SPLINE
SPL {X  -131.819, Y  +765.085, Z    +0.000, E1   -48.689, E3 +108359.963}
SPL {X  -153.047, Y  +721.053, Z    +0.000, E1   -34.410, E3 +108379.829}
SPL {X  -159.196, Y  +690.423, Z    +0.000, E1   -15.522, E3 +108384.926}
SPL {X  -160.000, Y  +672.957, Z    +0.000, E1    -0.766, E3 +108385.828}
SPL {X  -160.000, Y  +670.573, Z    +0.000, E1    +3.229, E3 +108385.856}
SPL {X  -160.000, Y  +665.683, Z    +0.000, E1   +13.339, E3 +108386.025}
SPL {X  -160.000, Y  +658.186, Z    +0.000, E1   +29.314, E3 +108386.629}
SPL {X  -160.000, Y  +642.169, Z    +0.000, E1   +52.097, E3 +108389.155}
SPL {X  -160.000, Y  +581.106, Z    +0.000, E1   +69.111, E3 +108410.027}
SPL {X  -160.000, Y  +418.281, Z    +0.000, E1   +71.209, E3 +108501.377}
SPL {X  -153.877, Y  +341.861, Z    +0.000, E1   +74.632, E3 +108514.790}
SPL {X  -152.649, Y  +337.758, Z    +0.000, E1   +72.728, E3 +108536.453}
SPL {X  -150.568, Y  +331.578, Z    +0.000, E1   +70.963, E3 +108556.379}
SPL {X  -147.367, Y  +323.387, Z    +0.000, E1   +69.846, E3 +108570.999}
SPL {X  -143.458, Y  +314.849, Z    +0.000, E1   +69.330, E3 +108580.881}
SPL {X  -137.919, Y  +304.592, Z    +0.000, E1   +68.645, E3 +108593.170}
SPL {X  -132.252, Y  +295.648, Z    +0.000, E1   +67.759, E3 +108604.485}
SPL {X  -127.852, Y  +289.504, Z    +0.000, E1   +67.080, E3 +108612.317}
SPL {X  -124.264, Y  +284.911, Z    +0.000, E1   +66.468, E3 +108618.213}
SPL {X   -87.531, Y  +251.766, Z    +0.000, E1   +54.242, E3 +108746.530}
ENDSPLINE

SPLINE
SPL {X  -130.414, Y  +293.006, Z    +0.000, E1   +48.816, E3 +108895.142}
SPL {X  -151.093, Y  +333.061, Z    +0.000, E1   +36.955, E3 +108916.423}
SPL {X  -158.896, Y  +366.939, Z    +0.000, E1   +17.535, E3 +108922.962}
SPL {X  -160.000, Y  +387.267, Z    +0.000, E1    +0.577, E3 +108924.152}
SPL {X  -160.000, Y  +391.471, Z    +0.000, E1    -7.208, E3 +108924.233}
SPL {X  -160.000, Y  +398.523, Z    +0.000, E1   -22.265, E3 +108924.645}
SPL {X  -160.000, Y  +411.325, Z    +0.000, E1   -44.857, E3 +108926.311}
SPL {X  -160.000, Y  +459.786, Z    +0.000, E1   -66.828, E3 +108941.704}
SPL {X  -160.000, Y  +650.407, Z    +0.000, E1   -71.387, E3 +109044.361}
SPL {X  -159.770, Y  +682.971, Z    +0.000, E1   -71.362, E3 +109067.936}
SPL {X  -156.288, Y  +708.665, Z    +0.000, E1   -70.996, E3 +109089.946}
SPL {X  -150.837, Y  +727.770, Z    +0.000, E1   -70.337, E3 +109109.280}
SPL {X  -144.661, Y  +742.760, Z    +0.000, E1   -69.570, E3 +109126.038}
SPL {X  -137.606, Y  +756.037, Z    +0.000, E1   -68.631, E3 +109142.003}
SPL {X  -131.907, Y  +764.957, Z    +0.000, E1   -67.736, E3 +109153.298}
SPL {X  -127.608, Y  +770.921, Z    +0.000, E1   -67.067, E3 +109160.917}
SPL {X  -124.072, Y  +775.426, Z    +0.000, E1   -66.459, E3 +109166.697}
SPL {X   -86.375, Y  +809.082, Z    +0.000, E1   -54.606, E3 +109291.027}
ENDSPLINE

SPLINE
SPL {X  -131.819, Y  +765.085, Z    +0.000, E1   -48.689, E3 +109446.921}
SPL {X  -153.047, Y  +721.053, Z    +0.000, E1   -34.410, E3 +109466.787}
SPL {X  -159.196, Y  +690.423, Z    +0.000, E1   -15.522, E3 +109471.883}
SPL {X  -160.000, Y  +672.957, Z    +0.000, E1    -0.766, E3 +109472.785}
SPL {X  -160.000, Y  +670.573, Z    +0.000, E1    +3.229, E3 +109472.813}
SPL {X  -160.000, Y  +665.683, Z    +0.000, E1   +13.339, E3 +109472.982}
SPL {X  -160.000, Y  +658.186, Z    +0.000, E1   +29.314, E3 +109473.586}
SPL {X  -160.000, Y  +642.169, Z    +0.000, E1   +52.097, E3 +109476.112}
SPL {X  -160.000, Y  +581.106, Z    +0.000, E1   +69.111, E3 +109496.984}
SPL {X  -160.000, Y  +418.281, Z    +0.000, E1   +71.209, E3 +109588.334}
SPL {X  -153.877, Y  +341.861, Z    +0.000, E1   +74.632, E3 +109601.747}
SPL {X  -152.649, Y  +337.758, Z    +0.000, E1   +72.728, E3 +109623.410}
SPL {X  -150.568, Y  +331.578, Z    +0.000, E1   +70.963, E3 +109643.336}
SPL {X  -147.367, Y  +323.387, Z    +0.000, E1   +69.846, E3 +109657.956}
SPL {X  -143.458, Y  +314.849, Z    +0.000, E1   +69.330, E3 +109667.839}
SPL {X  -137.919, Y  +304.592, Z    +0.000, E1   +68.645, E3 +109680.127}
SPL {X  -132.252, Y  +295.648, Z    +0.000, E1   +67.759, E3 +109691.442}
SPL {X  -127.852, Y  +289.504, Z    +0.000, E1   +67.080, E3 +109699.274}
SPL {X  -124.264, Y  +284.911, Z    +0.000, E1   +66.468, E3 +109705.170}
SPL {X   -87.531, Y  +251.766, Z    +0.000, E1   +54.242, E3 +109833.487}
ENDSPLINE

SPLINE
SPL {X  -130.414, Y  +293.006, Z    +0.000, E1   +48.816, E3 +109982.099}
SPL {X  -151.093, Y  +333.061, Z    +0.000, E1   +36.955, E3 +110003.380}
SPL {X  -158.896, Y  +366.939, Z    +0.000, E1   +17.535, E3 +110009.919}
SPL {X  -160.000, Y  +387.267, Z    +0.000, E1    +0.577, E3 +110011.109}
SPL {X  -160.000, Y  +391.471, Z    +0.000, E1    -7.208, E3 +110011.190}
SPL {X  -160.000, Y  +398.523, Z    +0.000, E1   -22.265, E3 +110011.602}
SPL {X  -160.000, Y  +411.325, Z    +0.000, E1   -44.857, E3 +110013.268}
SPL {X  -160.000, Y  +459.786, Z    +0.000, E1   -66.828, E3 +110028.661}
SPL {X  -160.000, Y  +650.407, Z    +0.000, E1   -71.387, E3 +110131.318}
SPL {X  -159.770, Y  +682.971, Z    +0.000, E1   -71.362, E3 +110154.893}
SPL {X  -156.288, Y  +708.665, Z    +0.000, E1   -70.996, E3 +110176.903}
SPL {X  -150.837, Y  +727.770, Z    +0.000, E1   -70.337, E3 +110196.237}
SPL {X  -144.661, Y  +742.760, Z    +0.000, E1   -69.570, E3 +110212.995}
SPL {X  -137.606, Y  +756.037, Z    +0.000, E1   -68.631, E3 +110228.960}
SPL {X  -131.907, Y  +764.957, Z    +0.000, E1   -67.736, E3 +110240.255}
SPL {X  -127.608, Y  +770.921, Z    +0.000, E1   -67.067, E3 +110247.874}
SPL {X  -124.072, Y  +775.426, Z    +0.000, E1   -66.459, E3 +110253.654}
SPL {X   -86.375, Y  +809.082, Z    +0.000, E1   -54.606, E3 +110377.984}
ENDSPLINE

SPLINE
SPL {X  -131.819, Y  +765.085, Z    +0.000, E1   -48.689, E3 +110533.878}
SPL {X  -153.047, Y  +721.053, Z    +0.000, E1   -34.410, E3 +110553.744}
SPL {X  -159.196, Y  +690.423, Z    +0.000, E1   -15.522, E3 +110558.840}
SPL {X  -160.000, Y  +672.957, Z    +0.000, E1    -0.766, E3 +110559.742}
SPL {X  -160.000, Y  +670.573, Z    +0.000, E1    +3.229, E3 +110559.770}
SPL {X  -160.000, Y  +665.683, Z    +0.000, E1   +13.339, E3 +110559.939}
SPL {X  -160.000, Y  +658.186, Z    +0.000, E1   +29.314, E3 +110560.544}
SPL {X  -160.000, Y  +642.169, Z    +0.000, E1   +52.097, E3 +110563.069}
SPL {X  -160.000, Y  +581.106, Z    +0.000, E1   +69.111, E3 +110583.941}
SPL {X  -160.000, Y  +418.281, Z    +0.000, E1   +71.209, E3 +110675.291}
SPL {X  -153.877, Y  +341.861, Z    +0.000, E1   +74.632, E3 +110688.704}
SPL {X  -152.649, Y  +337.758, Z    +0.000, E1   +72.728, E3 +110710.367}
SPL {X  -150.568, Y  +331.578, Z    +0.000, E1   +70.963, E3 +110730.293}
SPL {X  -147.367, Y  +323.387, Z    +0.000, E1   +69.846, E3 +110744.913}
SPL {X  -143.458, Y  +314.849, Z    +0.000, E1   +69.330, E3 +110754.796}
SPL {X  -137.919, Y  +304.592, Z    +0.000, E1   +68.645, E3 +110767.084}
SPL {X  -132.252, Y  +295.648, Z    +0.000, E1   +67.759, E3 +110778.399}
SPL {X  -127.852, Y  +289.504, Z    +0.000, E1   +67.080, E3 +110786.231}
SPL {X  -124.264, Y  +284.911, Z    +0.000, E1   +66.468, E3 +110792.127}
SPL {X   -87.531, Y  +251.766, Z    +0.000, E1   +54.242, E3 +110920.444}
ENDSPLINE

SPLINE
SPL {X  -130.414, Y  +293.006, Z    +0.000, E1   +48.816, E3 +111069.056}
SPL {X  -151.093, Y  +333.061, Z    +0.000, E1   +36.955, E3 +111090.337}
SPL {X  -158.896, Y  +366.939, Z    +0.000, E1   +17.535, E3 +111096.877}
SPL {X  -160.000, Y  +387.267, Z    +0.000, E1    +0.577, E3 +111098.066}
SPL {X  -160.000, Y  +391.471, Z    +0.000, E1    -7.208, E3 +111098.147}
SPL {X  -160.000, Y  +398.523, Z    +0.000, E1   -22.265, E3 +111098.559}
SPL {X  -160.000, Y  +411.325, Z    +0.000, E1   -44.857, E3 +111100.225}
SPL {X  -160.000, Y  +459.786, Z    +0.000, E1   -66.828, E3 +111115.618}
SPL {X  -160.000, Y  +650.407, Z    +0.000, E1   -71.387, E3 +111218.275}
SPL {X  -159.770, Y  +682.971, Z    +0.000, E1   -71.362, E3 +111241.850}
SPL {X  -156.288, Y  +708.665, Z    +0.000, E1   -70.996, E3 +111263.861}
SPL {X  -150.837, Y  +727.770, Z    +0.000, E1   -70.337, E3 +111283.194}
SPL {X  -144.661, Y  +742.760, Z    +0.000, E1   -69.570, E3 +111299.953}
SPL {X  -137.606, Y  +756.037, Z    +0.000, E1   -68.631, E3 +111315.917}
SPL {X  -131.907, Y  +764.957, Z    +0.000, E1   -67.736, E3 +111327.212}
SPL {X  -127.608, Y  +770.921, Z    +0.000, E1   -67.067, E3 +111334.831}
SPL {X  -124.072, Y  +775.426, Z    +0.000, E1   -66.459, E3 +111340.611}
SPL {X   -86.375, Y  +809.082, Z    +0.000, E1   -54.606, E3 +111464.941}
ENDSPLINE

SPLINE
SPL {X  -131.819, Y  +765.085, Z    +0.000, E1   -48.689, E3 +111620.835}
SPL {X  -153.047, Y  +721.053, Z    +0.000, E1   -34.410, E3 +111640.701}
SPL {X  -159.196, Y  +690.423, Z    +0.000, E1   -15.522, E3 +111645.797}
SPL {X  -160.000, Y  +672.957, Z    +0.000, E1    -0.766, E3 +111646.699}
SPL {X  -160.000, Y  +670.573, Z    +0.000, E1    +3.229, E3 +111646.727}
SPL {X  -160.000, Y  +665.683, Z    +0.000, E1   +13.339, E3 +111646.896}
SPL {X  -160.000, Y  +658.186, Z    +0.000, E1   +29.314, E3 +111647.501}
SPL {X  -160.000, Y  +642.169, Z    +0.000, E1   +52.097, E3 +111650.026}
SPL {X  -160.000, Y  +581.106, Z    +0.000, E1   +69.111, E3 +111670.898}
SPL {X  -160.000, Y  +418.281, Z    +0.000, E1   +71.209, E3 +111762.248}
SPL {X  -153.877, Y  +341.861, Z    +0.000, E1   +74.632, E3 +111775.662}
SPL {X  -152.649, Y  +337.758, Z    +0.000, E1   +72.728, E3 +111797.324}
SPL {X  -150.568, Y  +331.578, Z    +0.000, E1   +70.963, E3 +111817.250}
SPL {X  -147.367, Y  +323.387, Z    +0.000, E1   +69.846, E3 +111831.870}
SPL {X  -143.458, Y  +314.849, Z    +0.000, E1   +69.330, E3 +111841.753}
SPL {X  -137.919, Y  +304.592, Z    +0.000, E1   +68.645, E3 +111854.041}
SPL {X  -132.252, Y  +295.648, Z    +0.000, E1   +67.759, E3 +111865.356}
SPL {X  -127.852, Y  +289.504, Z    +0.000, E1   +67.080, E3 +111873.188}
SPL {X  -124.264, Y  +284.911, Z    +0.000, E1   +66.468, E3 +111879.084}
SPL {X   -87.531, Y  +251.766, Z    +0.000, E1   +54.242, E3 +112007.401}
ENDSPLINE

SPLINE
SPL {X  -130.414, Y  +293.006, Z    +0.000, E1   +48.816, E3 +112156.013}
SPL {X  -151.093, Y  +333.061, Z    +0.000, E1   +36.955, E3 +112177.294}
SPL {X  -158.896, Y  +366.939, Z    +0.000, E1   +17.535, E3 +112183.834}
SPL {X  -160.000, Y  +387.267, Z    +0.000, E1    +0.577, E3 +112185.024}
SPL {X  -160.000, Y  +391.471, Z    +0.000, E1    -7.208, E3 +112185.104}
SPL {X  -160.000, Y  +398.523, Z    +0.000, E1   -22.265, E3 +112185.516}
SPL {X  -160.000, Y  +411.325, Z    +0.000, E1   -44.857, E3 +112187.182}
SPL {X  -160.000, Y  +459.786, Z    +0.000, E1   -66.828, E3 +112202.575}
SPL {X  -160.000, Y  +650.407, Z    +0.000, E1   -71.387, E3 +112305.232}
SPL {X  -159.770, Y  +682.971, Z    +0.000, E1   -71.362, E3 +112328.807}
SPL {X  -156.288, Y  +708.665, Z    +0.000, E1   -70.996, E3 +112350.818}
SPL {X  -150.837, Y  +727.770, Z    +0.000, E1   -70.337, E3 +112370.151}
SPL {X  -144.661, Y  +742.760, Z    +0.000, E1   -69.570, E3 +112386.910}
SPL {X  -137.606, Y  +756.037, Z    +0.000, E1   -68.631, E3 +112402.874}
SPL {X  -131.907, Y  +764.957, Z    +0.000, E1   -67.736, E3 +112414.169}
SPL {X  -127.608, Y  +770.921, Z    +0.000, E1   -67.067, E3 +112421.788}
SPL {X  -124.072, Y  +775.426, Z    +0.000, E1   -66.459, E3 +112427.568}
SPL {X   -86.375, Y  +809.082, Z    +0.000, E1   -54.606, E3 +112551.898}
ENDSPLINE

SPLINE
SPL {X  -131.819, Y  +765.085, Z    +0.000, E1   -48.689, E3 +112707.792}
SPL {X  -153.047, Y  +721.053, Z    +0.000, E1   -34.410, E3 +112727.658}
SPL {X  -159.196, Y  +690.423, Z    +0.000, E1   -15.522, E3 +112732.754}
SPL {X  -160.000, Y  +672.957, Z    +0.000, E1    -0.766, E3 +112733.656}
SPL {X  -160.000, Y  +670.573, Z    +0.000, E1    +3.229, E3 +112733.684}
SPL {X  -160.000, Y  +665.683, Z    +0.000, E1   +13.339, E3 +112733.854}
SPL {X  -160.000, Y  +658.186, Z    +0.000, E1   +29.314, E3 +112734.458}
SPL {X  -160.000, Y  +642.169, Z    +0.000, E1   +52.097, E3 +112736.983}
SPL {X  -160.000, Y  +581.106, Z    +0.000, E1   +69.111, E3 +112757.856}
SPL {X  -160.000, Y  +418.281, Z    +0.000, E1   +71.209, E3 +112849.205}
SPL {X  -153.877, Y  +341.861, Z    +0.000, E1   +74.632, E3 +112862.619}
SPL {X  -152.649, Y  +337.758, Z    +0.000, E1   +72.728, E3 +112884.281}
SPL {X  -150.568, Y  +331.578, Z    +0.000, E1   +70.963, E3 +112904.207}
SPL {X  -147.367, Y  +323.387, Z    +0.000, E1   +69.846, E3 +112918.828}
SPL {X  -143.458, Y  +314.849, Z    +0.000, E1   +69.330, E3 +112928.710}
SPL {X  -137.919, Y  +304.592, Z    +0.000, E1   +68.645, E3 +112940.999}
SPL {X  -132.252, Y  +295.648, Z    +0.000, E1   +67.759, E3 +112952.313}
SPL {X  -127.852, Y  +289.504, Z    +0.000, E1   +67.080, E3 +112960.146}
SPL {X  -124.264, Y  +284.911, Z    +0.000, E1   +66.468, E3 +112966.041}
SPL {X   -87.531, Y  +251.766, Z    +0.000, E1   +54.242, E3 +113094.358}
ENDSPLINE

SPLINE
SPL {X  -130.414, Y  +293.006, Z    +0.000, E1   +48.816, E3 +113242.971}
SPL {X  -151.093, Y  +333.061, Z    +0.000, E1   +36.955, E3 +113264.251}
SPL {X  -158.896, Y  +366.939, Z    +0.000, E1   +17.535, E3 +113270.791}
SPL {X  -160.000, Y  +387.267, Z    +0.000, E1    +0.577, E3 +113271.981}
SPL {X  -160.000, Y  +391.471, Z    +0.000, E1    -7.208, E3 +113272.062}
SPL {X  -160.000, Y  +398.523, Z    +0.000, E1   -22.265, E3 +113272.473}
SPL {X  -160.000, Y  +411.325, Z    +0.000, E1   -44.857, E3 +113274.139}
SPL {X  -160.000, Y  +459.786, Z    +0.000, E1   -66.828, E3 +113289.532}
SPL {X  -160.000, Y  +650.407, Z    +0.000, E1   -71.387, E3 +113392.189}
SPL {X  -159.770, Y  +682.971, Z    +0.000, E1   -71.362, E3 +113415.765}
SPL {X  -156.288, Y  +708.665, Z    +0.000, E1   -70.996, E3 +113437.775}
SPL {X  -150.837, Y  +727.770, Z    +0.000, E1   -70.337, E3 +113457.108}
SPL {X  -144.661, Y  +742.760, Z    +0.000, E1   -69.570, E3 +113473.867}
SPL {X  -137.606, Y  +756.037, Z    +0.000, E1   -68.631, E3 +113489.831}
SPL {X  -131.907, Y  +764.957, Z    +0.000, E1   -67.736, E3 +113501.126}
SPL {X  -127.608, Y  +770.921, Z    +0.000, E1   -67.067, E3 +113508.745}
SPL {X  -124.072, Y  +775.426, Z    +0.000, E1   -66.459, E3 +113514.525}
SPL {X   -86.375, Y  +809.082, Z    +0.000, E1   -54.606, E3 +113638.856}
ENDSPLINE

SPLINE
SPL {X  -131.819, Y  +765.085, Z    +0.000, E1   -48.689, E3 +113794.749}
SPL {X  -153.047, Y  +721.053, Z    +0.000, E1   -34.410, E3 +113814.615}
SPL {X  -159.196, Y  +690.423, Z    +0.000, E1   -15.522, E3 +113819.711}
SPL {X  -160.000, Y  +672.957, Z    +0.000, E1    -0.766, E3 +113820.613}
SPL {X  -160.000, Y  +670.573, Z    +0.000, E1    +3.229, E3 +113820.641}
SPL {X  -160.000, Y  +665.683, Z    +0.000, E1   +13.339, E3 +113820.811}
SPL {X  -160.000, Y  +658.186, Z    +0.000, E1   +29.314, E3 +113821.415}
SPL {X  -160.000, Y  +642.169, Z    +0.000, E1   +52.097, E3 +113823.940}
SPL {X  -160.000, Y  +581.106, Z    +0.000, E1   +69.111, E3 +113844.813}
SPL {X  -160.000, Y  +418.281, Z    +0.000, E1   +71.209, E3 +113936.162}
SPL {X  -153.877, Y  +341.861, Z    +0.000, E1   +74.632, E3 +113949.576}
SPL {X  -152.649, Y  +337.758, Z    +0.000, E1   +72.728, E3 +113971.238}
SPL {X  -150.568, Y  +331.578, Z    +0.000, E1   +70.963, E3 +113991.164}
SPL {X  -147.367, Y  +323.387, Z    +0.000, E1   +69.846, E3 +114005.785}
SPL {X  -143.458, Y  +314.849, Z    +0.000, E1   +69.330, E3 +114015.667}
SPL {X  -137.919, Y  +304.592, Z    +0.000, E1   +68.645, E3 +114027.956}
SPL {X  -132.252, Y  +295.648, Z    +0.000, E1   +67.759, E3 +114039.270}
SPL {X  -127.852, Y  +289.504, Z    +0.000, E1   +67.080, E3 +114047.103}
SPL {X  -124.264, Y  +284.911, Z    +0.000, E1   +66.468, E3 +114052.999}
SPL {X   -87.531, Y  +251.766, Z    +0.000, E1   +54.242, E3 +114181.315}
ENDSPLINE

SPLINE
SPL {X  -130.414, Y  +293.006, Z    +0.000, E1   +48.816, E3 +114329.928}
SPL {X  -151.093, Y  +333.061, Z    +0.000, E1   +36.955, E3 +114351.208}
SPL {X  -158.896, Y  +366.939, Z    +0.000, E1   +17.535, E3 +114357.748}
SPL {X  -160.000, Y  +387.267, Z    +0.000, E1    +0.577, E3 +114358.938}
SPL {X  -160.000, Y  +391.471, Z    +0.000, E1    -7.208, E3 +114359.019}
SPL {X  -160.000, Y  +398.523, Z    +0.000, E1   -22.265, E3 +114359.431}
SPL {X  -160.000, Y  +411.325, Z    +0.000, E1   -44.857, E3 +114361.096}
SPL {X  -160.000, Y  +459.786, Z    +0.000, E1   -66.828, E3 +114376.489}
SPL {X  -160.000, Y  +650.407, Z    +0.000, E1   -71.387, E3 +114479.146}
SPL {X  -159.770, Y  +682.971, Z    +0.000, E1   -71.362, E3 +114502.722}
SPL {X  -156.288, Y  +708.665, Z    +0.000, E1   -70.996, E3 +114524.732}
SPL {X  -150.837, Y  +727.770, Z    +0.000, E1   -70.337, E3 +114544.066}
SPL {X  -144.661, Y  +742.760, Z    +0.000, E1   -69.570, E3 +114560.824}
SPL {X  -137.606, Y  +756.037, Z    +0.000, E1   -68.631, E3 +114576.789}
SPL {X  -131.907, Y  +764.957, Z    +0.000, E1   -67.736, E3 +114588.084}
SPL {X  -127.608, Y  +770.921, Z    +0.000, E1   -67.067, E3 +114595.702}
SPL {X  -124.072, Y  +775.426, Z    +0.000, E1   -66.459, E3 +114601.482}
SPL {X   -86.375, Y  +809.082, Z    +0.000, E1   -54.606, E3 +114725.813}
ENDSPLINE

SPLINE
SPL {X  -131.819, Y  +765.085, Z    +0.000, E1   -48.689, E3 +114881.706}
SPL {X  -153.047, Y  +721.053, Z    +0.000, E1   -34.410, E3 +114901.572}
SPL {X  -159.196, Y  +690.423, Z    +0.000, E1   -15.522, E3 +114906.669}
SPL {X  -160.000, Y  +672.957, Z    +0.000, E1    -0.766, E3 +114907.570}
SPL {X  -160.000, Y  +670.573, Z    +0.000, E1    +3.229, E3 +114907.599}
SPL {X  -160.000, Y  +665.683, Z    +0.000, E1   +13.339, E3 +114907.768}
SPL {X  -160.000, Y  +658.186, Z    +0.000, E1   +29.314, E3 +114908.372}
SPL {X  -160.000, Y  +642.169, Z    +0.000, E1   +52.097, E3 +114910.898}
SPL {X  -160.000, Y  +581.106, Z    +0.000, E1   +69.111, E3 +114931.770}
SPL {X  -160.000, Y  +418.281, Z    +0.000, E1   +71.209, E3 +115023.119}
SPL {X  -153.877, Y  +341.861, Z    +0.000, E1   +74.632, E3 +115036.533}
SPL {X  -152.649, Y  +337.758, Z    +0.000, E1   +72.728, E3 +115058.196}
SPL {X  -150.568, Y  +331.578, Z    +0.000, E1   +70.963, E3 +115078.121}
SPL {X  -147.367, Y  +323.387, Z    +0.000, E1   +69.846, E3 +115092.742}
SPL {X  -143.458, Y  +314.849, Z    +0.000, E1   +69.330, E3 +115102.624}
SPL {X  -137.919, Y  +304.592, Z    +0.000, E1   +68.645, E3 +115114.913}
SPL {X  -132.252, Y  +295.648, Z    +0.000, E1   +67.759, E3 +115126.228}
SPL {X  -127.852, Y  +289.504, Z    +0.000, E1   +67.080, E3 +115134.060}
SPL {X  -124.264, Y  +284.911, Z    +0.000, E1   +66.468, E3 +115139.956}
SPL {X   -87.531, Y  +251.766, Z    +0.000, E1   +54.242, E3 +115268.272}
ENDSPLINE

SPLINE
SPL {X  -130.414, Y  +293.006, Z    +0.000, E1   +48.816, E3 +115416.885}
SPL {X  -151.093, Y  +333.061, Z    +0.000, E1   +36.955, E3 +115438.165}
SPL {X  -158.896, Y  +366.939, Z    +0.000, E1   +17.535, E3 +115444.705}
SPL {X  -160.000, Y  +387.267, Z    +0.000, E1    +0.577, E3 +115445.895}
SPL {X  -160.000, Y  +391.471, Z    +0.000, E1    -7.208, E3 +115445.976}
SPL {X  -160.000, Y  +398.523, Z    +0.000, E1   -22.265, E3 +115446.388}
SPL {X  -160.000, Y  +411.325, Z    +0.000, E1   -44.857, E3 +115448.054}
SPL {X  -160.000, Y  +459.786, Z    +0.000, E1   -66.828, E3 +115463.446}
SPL {X  -160.000, Y  +650.407, Z    +0.000, E1   -71.387, E3 +115566.103}
SPL {X  -159.770, Y  +682.971, Z    +0.000, E1   -71.362, E3 +115589.679}
SPL {X  -156.288, Y  +708.665, Z    +0.000, E1   -70.996, E3 +115611.689}
SPL {X  -150.837, Y  +727.770, Z    +0.000, E1   -70.337, E3 +115631.023}
SPL {X  -144.661, Y  +742.760, Z    +0.000, E1   -69.570, E3 +115647.781}
SPL {X  -137.606, Y  +756.037, Z    +0.000, E1   -68.631, E3 +115663.746}
SPL {X  -131.907, Y  +764.957, Z    +0.000, E1   -67.736, E3 +115675.041}
SPL {X  -127.608, Y  +770.921, Z    +0.000, E1   -67.067, E3 +115682.659}
SPL {X  -124.072, Y  +775.426, Z    +0.000, E1   -66.459, E3 +115688.440}
SPL {X   -86.375, Y  +809.082, Z    +0.000, E1   -54.606, E3 +115812.770}
ENDSPLINE

SPLINE
SPL {X  -131.819, Y  +765.085, Z    +0.000, E1   -48.689, E3 +115968.663}
SPL {X  -153.047, Y  +721.053, Z    +0.000, E1   -34.410, E3 +115988.529}
SPL {X  -159.196, Y  +690.423, Z    +0.000, E1   -15.522, E3 +115993.626}
SPL {X  -160.000, Y  +672.957, Z    +0.000, E1    -0.766, E3 +115994.528}
SPL {X  -160.000, Y  +670.573, Z    +0.000, E1    +3.229, E3 +115994.556}
SPL {X  -160.000, Y  +665.683, Z    +0.000, E1   +13.339, E3 +115994.725}
SPL {X  -160.000, Y  +658.186, Z    +0.000, E1   +29.314, E3 +115995.329}
SPL {X  -160.000, Y  +642.169, Z    +0.000, E1   +52.097, E3 +115997.855}
SPL {X  -160.000, Y  +581.106, Z    +0.000, E1   +69.111, E3 +116018.727}
SPL {X  -160.000, Y  +418.281, Z    +0.000, E1   +71.209, E3 +116110.076}
SPL {X  -153.877, Y  +341.861, Z    +0.000, E1   +74.632, E3 +116123.490}
SPL {X  -152.649, Y  +337.758, Z    +0.000, E1   +72.728, E3 +116145.153}
SPL {X  -150.568, Y  +331.578, Z    +0.000, E1   +70.963, E3 +116165.079}
SPL {X  -147.367, Y  +323.387, Z    +0.000, E1   +69.846, E3 +116179.699}
SPL {X  -143.458, Y  +314.849, Z    +0.000, E1   +69.330, E3 +116189.581}
SPL {X  -137.919, Y  +304.592, Z    +0.000, E1   +68.645, E3 +116201.870}
SPL {X  -132.252, Y  +295.648, Z    +0.000, E1   +67.759, E3 +116213.185}
SPL {X  -127.852, Y  +289.504, Z    +0.000, E1   +67.080, E3 +116221.017}
SPL {X  -124.264, Y  +284.911, Z    +0.000, E1   +66.468, E3 +116226.913}
SPL {X   -87.531, Y  +251.766, Z    +0.000, E1   +54.242, E3 +116355.229}
ENDSPLINE

SPLINE
SPL {X  -130.414, Y  +293.006, Z    +0.000, E1   +48.816, E3 +116503.842}
SPL {X  -151.093, Y  +333.061, Z    +0.000, E1   +36.955, E3 +116525.122}
SPL {X  -158.896, Y  +366.939, Z    +0.000, E1   +17.535, E3 +116531.662}
SPL {X  -160.000, Y  +387.267, Z    +0.000, E1    +0.577, E3 +116532.852}
SPL {X  -160.000, Y  +391.471, Z    +0.000, E1    -7.208, E3 +116532.933}
SPL {X  -160.000, Y  +398.523, Z    +0.000, E1   -22.265, E3 +116533.345}
SPL {X  -160.000, Y  +411.325, Z    +0.000, E1   -44.857, E3 +116535.011}
SPL {X  -160.000, Y  +459.786, Z    +0.000, E1   -66.828, E3 +116550.403}
SPL {X  -160.000, Y  +650.407, Z    +0.000, E1   -71.387, E3 +116653.060}
SPL {X  -159.770, Y  +682.971, Z    +0.000, E1   -71.362, E3 +116676.636}
SPL {X  -156.288, Y  +708.665, Z    +0.000, E1   -70.996, E3 +116698.646}
SPL {X  -150.837, Y  +727.770, Z    +0.000, E1   -70.337, E3 +116717.980}
SPL {X  -144.661, Y  +742.760, Z    +0.000, E1   -69.570, E3 +116734.738}
SPL {X  -137.606, Y  +756.037, Z    +0.000, E1   -68.631, E3 +116750.703}
SPL {X  -131.907, Y  +764.957, Z    +0.000, E1   -67.736, E3 +116761.998}
SPL {X  -127.608, Y  +770.921, Z    +0.000, E1   -67.067, E3 +116769.616}
SPL {X  -124.072, Y  +775.426, Z    +0.000, E1   -66.459, E3 +116775.397}
SPL {X   -86.375, Y  +809.082, Z    +0.000, E1   -54.606, E3 +116899.727}
ENDSPLINE

SPLINE
SPL {X  -131.819, Y  +765.085, Z    +0.000, E1   -48.689, E3 +117055.620}
SPL {X  -153.047, Y  +721.053, Z    +0.000, E1   -34.410, E3 +117075.486}
SPL {X  -159.196, Y  +690.423, Z    +0.000, E1   -15.522, E3 +117080.583}
SPL {X  -160.000, Y  +672.957, Z    +0.000, E1    -0.766, E3 +117081.485}
SPL {X  -160.000, Y  +670.573, Z    +0.000, E1    +3.229, E3 +117081.513}
SPL {X  -160.000, Y  +665.683, Z    +0.000, E1   +13.339, E3 +117081.682}
SPL {X  -160.000, Y  +658.186, Z    +0.000, E1   +29.314, E3 +117082.286}
SPL {X  -160.000, Y  +642.169, Z    +0.000, E1   +52.097, E3 +117084.812}
SPL {X  -160.000, Y  +581.106, Z    +0.000, E1   +69.111, E3 +117105.684}
SPL {X  -160.000, Y  +418.281, Z    +0.000, E1   +71.209, E3 +117197.034}
SPL {X  -153.877, Y  +341.861, Z    +0.000, E1   +74.632, E3 +117210.447}
SPL {X  -152.649, Y  +337.758, Z    +0.000, E1   +72.728, E3 +117232.110}
SPL {X  -150.568, Y  +331.578, Z    +0.000, E1   +70.963, E3 +117252.036}
SPL {X  -147.367, Y  +323.387, Z    +0.000, E1   +69.846, E3 +117266.656}
SPL {X  -143.458, Y  +314.849, Z    +0.000, E1   +69.330, E3 +117276.538}
SPL {X  -137.919, Y  +304.592, Z    +0.000, E1   +68.645, E3 +117288.827}
SPL {X  -132.252, Y  +295.648, Z    +0.000, E1   +67.759, E3 +117300.142}
SPL {X  -127.852, Y  +289.504, Z    +0.000, E1   +67.080, E3 +117307.974}
SPL {X  -124.264, Y  +284.911, Z    +0.000, E1   +66.468, E3 +117313.870}
SPL {X   -87.531, Y  +251.766, Z    +0.000, E1   +54.242, E3 +117442.187}
ENDSPLINE

SPLINE
SPL {X  -130.414, Y  +293.006, Z    +0.000, E1   +48.816, E3 +117590.799}
SPL {X  -151.093, Y  +333.061, Z    +0.000, E1   +36.955, E3 +117612.080}
SPL {X  -158.896, Y  +366.939, Z    +0.000, E1   +17.535, E3 +117618.619}
SPL {X  -160.000, Y  +387.267, Z    +0.000, E1    +0.577, E3 +117619.809}
SPL {X  -160.000, Y  +391.471, Z    +0.000, E1    -7.208, E3 +117619.890}
SPL {X  -160.000, Y  +398.523, Z    +0.000, E1   -22.265, E3 +117620.302}
SPL {X  -160.000, Y  +411.325, Z    +0.000, E1   -44.857, E3 +117621.968}
SPL {X  -160.000, Y  +459.786, Z    +0.000, E1   -66.828, E3 +117637.361}
SPL {X  -160.000, Y  +650.407, Z    +0.000, E1   -71.387, E3 +117740.018}
SPL {X  -159.770, Y  +682.971, Z    +0.000, E1   -71.362, E3 +117763.593}
SPL {X  -156.288, Y  +708.665, Z    +0.000, E1   -70.996, E3 +117785.603}
SPL {X  -150.837, Y  +727.770, Z    +0.000, E1   -70.337, E3 +117804.937}
SPL {X  -144.661, Y  +742.760, Z    +0.000, E1   -69.570, E3 +117821.695}
SPL {X  -137.606, Y  +756.037, Z    +0.000, E1   -68.631, E3 +117837.660}
SPL {X  -131.907, Y  +764.957, Z    +0.000, E1   -67.736, E3 +117848.955}
SPL {X  -127.608, Y  +770.921, Z    +0.000, E1   -67.067, E3 +117856.573}
SPL {X  -124.072, Y  +775.426, Z    +0.000, E1   -66.459, E3 +117862.354}
SPL {X   -86.375, Y  +809.082, Z    +0.000, E1   -54.606, E3 +117986.684}
ENDSPLINE

SPLINE
SPL {X  -131.819, Y  +765.085, Z    +0.000, E1   -48.689, E3 +118142.577}
SPL {X  -153.047, Y  +721.053, Z    +0.000, E1   -34.410, E3 +118162.443}
SPL {X  -159.196, Y  +690.423, Z    +0.000, E1   -15.522, E3 +118167.540}
SPL {X  -160.000, Y  +672.957, Z    +0.000, E1    -0.766, E3 +118168.442}
SPL {X  -160.000, Y  +670.573, Z    +0.000, E1    +3.229, E3 +118168.470}
SPL {X  -160.000, Y  +665.683, Z    +0.000, E1   +13.339, E3 +118168.639}
SPL {X  -160.000, Y  +658.186, Z    +0.000, E1   +29.314, E3 +118169.243}
SPL {X  -160.000, Y  +642.169, Z    +0.000, E1   +52.097, E3 +118171.769}
SPL {X  -160.000, Y  +581.106, Z    +0.000, E1   +69.111, E3 +118192.641}
SPL {X  -160.000, Y  +418.281, Z    +0.000, E1   +71.209, E3 +118283.991}
SPL {X  -153.877, Y  +341.861, Z    +0.000, E1   +74.632, E3 +118297.404}
SPL {X  -152.649, Y  +337.758, Z    +0.000, E1   +72.728, E3 +118319.067}
SPL {X  -150.568, Y  +331.578, Z    +0.000, E1   +70.963, E3 +118338.993}
SPL {X  -147.367, Y  +323.387, Z    +0.000, E1   +69.846, E3 +118353.613}
SPL {X  -143.458, Y  +314.849, Z    +0.000, E1   +69.330, E3 +118363.495}
SPL {X  -137.919, Y  +304.592, Z    +0.000, E1   +68.645, E3 +118375.784}
SPL {X  -132.252, Y  +295.648, Z    +0.000, E1   +67.759, E3 +118387.099}
SPL {X  -127.852, Y  +289.504, Z    +0.000, E1   +67.080, E3 +118394.931}
SPL {X  -124.264, Y  +284.911, Z    +0.000, E1   +66.468, E3 +118400.827}
SPL {X   -87.531, Y  +251.766, Z    +0.000, E1   +54.242, E3 +118529.144}
ENDSPLINE

SPLINE
SPL {X  -130.414, Y  +293.006, Z    +0.000, E1   +48.816, E3 +118677.756}
SPL {X  -151.093, Y  +333.061, Z    +0.000, E1   +36.955, E3 +118699.037}
SPL {X  -158.896, Y  +366.939, Z    +0.000, E1   +17.535, E3 +118705.576}
SPL {X  -160.000, Y  +387.267, Z    +0.000, E1    +0.577, E3 +118706.766}
SPL {X  -160.000, Y  +391.471, Z    +0.000, E1    -7.208, E3 +118706.847}
SPL {X  -160.000, Y  +398.523, Z    +0.000, E1   -22.265, E3 +118707.259}
SPL {X  -160.000, Y  +411.325, Z    +0.000, E1   -44.857, E3 +118708.925}
SPL {X  -160.000, Y  +459.786, Z    +0.000, E1   -66.828, E3 +118724.318}
SPL {X  -160.000, Y  +650.407, Z    +0.000, E1   -71.387, E3 +118826.975}
SPL {X  -159.770, Y  +682.971, Z    +0.000, E1   -71.362, E3 +118850.550}
SPL {X  -156.288, Y  +708.665, Z    +0.000, E1   -70.996, E3 +118872.560}
SPL {X  -150.837, Y  +727.770, Z    +0.000, E1   -70.337, E3 +118891.894}
SPL {X  -144.661, Y  +742.760, Z    +0.000, E1   -69.570, E3 +118908.652}
SPL {X  -137.606, Y  +756.037, Z    +0.000, E1   -68.631, E3 +118924.617}
SPL {X  -131.907, Y  +764.957, Z    +0.000, E1   -67.736, E3 +118935.912}
SPL {X  -127.608, Y  +770.921, Z    +0.000, E1   -67.067, E3 +118943.531}
SPL {X  -124.072, Y  +775.426, Z    +0.000, E1   -66.459, E3 +118949.311}
SPL {X   -86.375, Y  +809.082, Z    +0.000, E1   -54.606, E3 +119073.641}
ENDSPLINE

SPLINE
SPL {X  -131.819, Y  +765.085, Z    +0.000, E1   -48.689, E3 +119229.535}
SPL {X  -153.047, Y  +721.053, Z    +0.000, E1   -34.410, E3 +119249.401}
SPL {X  -159.196, Y  +690.423, Z    +0.000, E1   -15.522, E3 +119254.497}
SPL {X  -160.000, Y  +672.957, Z    +0.000, E1    -0.766, E3 +119255.399}
SPL {X  -160.000, Y  +670.573, Z    +0.000, E1    +3.229, E3 +119255.427}
SPL {X  -160.000, Y  +665.683, Z    +0.000, E1   +13.339, E3 +119255.596}
SPL {X  -160.000, Y  +658.186, Z    +0.000, E1   +29.314, E3 +119256.200}
SPL {X  -160.000, Y  +642.169, Z    +0.000, E1   +52.097, E3 +119258.726}
SPL {X  -160.000, Y  +581.106, Z    +0.000, E1   +69.111, E3 +119279.598}
SPL {X  -160.000, Y  +418.281, Z    +0.000, E1   +71.209, E3 +119370.948}
SPL {X  -153.877, Y  +341.861, Z    +0.000, E1   +74.632, E3 +119384.361}
SPL {X  -152.649, Y  +337.758, Z    +0.000, E1   +72.728, E3 +119406.024}
SPL {X  -150.568, Y  +331.578, Z    +0.000, E1   +70.963, E3 +119425.950}
SPL {X  -147.367, Y  +323.387, Z    +0.000, E1   +69.846, E3 +119440.570}
SPL {X  -143.458, Y  +314.849, Z    +0.000, E1   +69.330, E3 +119450.453}
SPL {X  -137.919, Y  +304.592, Z    +0.000, E1   +68.645, E3 +119462.741}
SPL {X  -132.252, Y  +295.648, Z    +0.000, E1   +67.759, E3 +119474.056}
SPL {X  -127.852, Y  +289.504, Z    +0.000, E1   +67.080, E3 +119481.888}
SPL {X  -124.264, Y  +284.911, Z    +0.000, E1   +66.468, E3 +119487.784}
SPL {X   -87.531, Y  +251.766, Z    +0.000, E1   +54.242, E3 +119616.101}
ENDSPLINE

SPLINE
SPL {X  -130.414, Y  +293.006, Z    +0.000, E1   +48.816, E3 +119764.713}
SPL {X  -151.093, Y  +333.061, Z    +0.000, E1   +36.955, E3 +119785.994}
SPL {X  -158.896, Y  +366.939, Z    +0.000, E1   +17.535, E3 +119792.534}
SPL {X  -160.000, Y  +387.267, Z    +0.000, E1    +0.577, E3 +119793.723}
SPL {X  -160.000, Y  +391.471, Z    +0.000, E1    -7.208, E3 +119793.804}
SPL {X  -160.000, Y  +398.523, Z    +0.000, E1   -22.265, E3 +119794.216}
SPL {X  -160.000, Y  +411.325, Z    +0.000, E1   -44.857, E3 +119795.882}
SPL {X  -160.000, Y  +459.786, Z    +0.000, E1   -66.828, E3 +119811.275}
SPL {X  -160.000, Y  +650.407, Z    +0.000, E1   -71.387, E3 +119913.932}
SPL {X  -159.770, Y  +682.971, Z    +0.000, E1   -71.362, E3 +119937.507}
SPL {X  -156.288, Y  +708.665, Z    +0.000, E1   -70.996, E3 +119959.517}
SPL {X  -150.837, Y  +727.770, Z    +0.000, E1   -70.337, E3 +119978.851}
SPL {X  -144.661, Y  +742.760, Z    +0.000, E1   -69.570, E3 +119995.609}
SPL {X  -137.606, Y  +756.037, Z    +0.000, E1   -68.631, E3 +120011.574}
SPL {X  -131.907, Y  +764.957, Z    +0.000, E1   -67.736, E3 +120022.869}
SPL {X  -127.608, Y  +770.921, Z    +0.000, E1   -67.067, E3 +120030.488}
SPL {X  -124.072, Y  +775.426, Z    +0.000, E1   -66.459, E3 +120036.268}
SPL {X   -86.375, Y  +809.082, Z    +0.000, E1   -54.606, E3 +120160.598}
ENDSPLINE

SPLINE
SPL {X  -131.819, Y  +765.085, Z    +0.000, E1   -48.689, E3 +120316.492}
SPL {X  -153.047, Y  +721.053, Z    +0.000, E1   -34.410, E3 +120336.358}
SPL {X  -159.196, Y  +690.423, Z    +0.000, E1   -15.522, E3 +120341.454}
SPL {X  -160.000, Y  +672.957, Z    +0.000, E1    -0.766, E3 +120342.356}
SPL {X  -160.000, Y  +670.573, Z    +0.000, E1    +3.229, E3 +120342.384}
SPL {X  -160.000, Y  +665.683, Z    +0.000, E1   +13.339, E3 +120342.553}
SPL {X  -160.000, Y  +658.186, Z    +0.000, E1   +29.314, E3 +120343.158}
SPL {X  -160.000, Y  +642.169, Z    +0.000, E1   +52.097, E3 +120345.683}
SPL {X  -160.000, Y  +581.106, Z    +0.000, E1   +69.111, E3 +120366.555}
SPL {X  -160.000, Y  +418.281, Z    +0.000, E1   +71.209, E3 +120457.905}
SPL {X  -153.877, Y  +341.861, Z    +0.000, E1   +74.632, E3 +120471.319}
SPL {X  -152.649, Y  +337.758, Z    +0.000, E1   +72.728, E3 +120492.981}
SPL {X  -150.568, Y  +331.578, Z    +0.000, E1   +70.963, E3 +120512.907}
SPL {X  -147.367, Y  +323.387, Z    +0.000, E1   +69.846, E3 +120527.527}
SPL {X  -143.458, Y  +314.849, Z    +0.000, E1   +69.330, E3 +120537.410}
SPL {X  -137.919, Y  +304.592, Z    +0.000, E1   +68.645, E3 +120549.698}
SPL {X  -132.252, Y  +295.648, Z    +0.000, E1   +67.759, E3 +120561.013}
SPL {X  -127.852, Y  +289.504, Z    +0.000, E1   +67.080, E3 +120568.845}
SPL {X  -124.264, Y  +284.911, Z    +0.000, E1   +66.468, E3 +120574.741}
SPL {X   -87.531, Y  +251.766, Z    +0.000, E1   +54.242, E3 +120703.058}
ENDSPLINE

SPLINE
SPL {X  -130.414, Y  +293.006, Z    +0.000, E1   +48.816, E3 +120851.670}
SPL {X  -151.093, Y  +333.061, Z    +0.000, E1   +36.955, E3 +120872.951}
SPL {X  -158.896, Y  +366.939, Z    +0.000, E1   +17.535, E3 +120879.491}
SPL {X  -160.000, Y  +387.267, Z    +0.000, E1    +0.577, E3 +120880.680}
SPL {X  -160.000, Y  +391.471, Z    +0.000, E1    -7.208, E3 +120880.761}
SPL {X  -160.000, Y  +398.523, Z    +0.000, E1   -22.265, E3 +120881.173}
SPL {X  -160.000, Y  +411.325, Z    +0.000, E1   -44.857, E3 +120882.839}
SPL {X  -160.000, Y  +459.786, Z    +0.000, E1   -66.828, E3 +120898.232}
SPL {X  -160.000, Y  +650.407, Z    +0.000, E1   -71.387, E3 +121000.889}
SPL {X  -159.770, Y  +682.971, Z    +0.000, E1   -71.362, E3 +121024.464}
SPL {X  -156.288, Y  +708.665, Z    +0.000, E1   -70.996, E3 +121046.475}
SPL {X  -150.837, Y  +727.770, Z    +0.000, E1   -70.337, E3 +121065.808}
SPL {X  -144.661, Y  +742.760, Z    +0.000, E1   -69.570, E3 +121082.567}
SPL {X  -137.606, Y  +756.037, Z    +0.000, E1   -68.631, E3 +121098.531}
SPL {X  -131.907, Y  +764.957, Z    +0.000, E1   -67.736, E3 +121109.826}
SPL {X  -127.608, Y  +770.921, Z    +0.000, E1   -67.067, E3 +121117.445}
SPL {X  -124.072, Y  +775.426, Z    +0.000, E1   -66.459, E3 +121123.225}
SPL {X   -86.375, Y  +809.082, Z    +0.000, E1   -54.606, E3 +121247.555}
ENDSPLINE

SPLINE
SPL {X  -131.819, Y  +765.085, Z    +0.000, E1   -48.689, E3 +121403.449}
SPL {X  -153.047, Y  +721.053, Z    +0.000, E1   -34.410, E3 +121423.315}
SPL {X  -159.196, Y  +690.423, Z    +0.000, E1   -15.522, E3 +121428.411}
SPL {X  -160.000, Y  +672.957, Z    +0.000, E1    -0.766, E3 +121429.313}
SPL {X  -160.000, Y  +670.573, Z    +0.000, E1    +3.229, E3 +121429.341}
SPL {X  -160.000, Y  +665.683, Z    +0.000, E1   +13.339, E3 +121429.511}
SPL {X  -160.000, Y  +658.186, Z    +0.000, E1   +29.314, E3 +121430.115}
SPL {X  -160.000, Y  +642.169, Z    +0.000, E1   +52.097, E3 +121432.640}
SPL {X  -160.000, Y  +581.106, Z    +0.000, E1   +69.111, E3 +121453.513}
SPL {X  -160.000, Y  +418.281, Z    +0.000, E1   +71.209, E3 +121544.862}
SPL {X  -153.877, Y  +341.861, Z    +0.000, E1   +74.632, E3 +121558.276}
SPL {X  -152.649, Y  +337.758, Z    +0.000, E1   +72.728, E3 +121579.938}
SPL {X  -150.568, Y  +331.578, Z    +0.000, E1   +70.963, E3 +121599.864}
ENDSPLINE

SPLINE
SPL {X  -150.729, Y  +332.027, Z    +0.000, E1   +68.788, E3 +121616.733}
SPL {X  -146.876, Y  +322.238, Z    +0.000, E1   +68.294, E3 +121628.100}
SPL {X  -142.952, Y  +313.834, Z    +0.000, E1   +67.744, E3 +121638.379}
SPL {X  -139.245, Y  +306.891, Z    +0.000, E1   +67.208, E3 +121647.163}
SPL {X  -135.108, Y  +299.992, Z    +0.000, E1   +66.599, E3 +121656.114}
SPL {X  -130.642, Y  +293.328, Z    +0.000, E1   +65.888, E3 +121664.966}
SPL {X  -126.461, Y  +287.682, Z    +0.000, E1   +65.179, E3 +121672.529}
SPL {X   -93.259, Y  +255.690, Z    +0.000, E1   +54.095, E3 +121787.911}
ENDSPLINE

SPLINE
SPL {X  -130.811, Y  +293.568, Z    +0.000, E1   +46.951, E3 +121931.772}
SPL {X  -151.580, Y  +334.479, Z    +0.000, E1   +34.520, E3 +121955.894}
SPL {X  -157.897, Y  +359.846, Z    +0.000, E1   +21.040, E3 +121961.852}
SPL {X  -159.671, Y  +375.443, Z    +0.000, E1   +10.084, E3 +121963.667}
SPL {X  -160.000, Y  +387.403, Z    +0.000, E1    +0.377, E3 +121964.143}
SPL {X  -160.000, Y  +391.807, Z    +0.000, E1    -7.102, E3 +121964.247}
SPL {X  -160.000, Y  +398.244, Z    +0.000, E1   -19.803, E3 +121964.681}
SPL {X  -160.000, Y  +410.795, Z    +0.000, E1   -41.112, E3 +121966.494}
SPL {X  -160.000, Y  +461.796, Z    +0.000, E1   -65.564, E3 +121983.137}
SPL {X  -160.000, Y  +623.854, Z    +0.000, E1   -69.845, E3 +122077.209}
SPL {X  -160.000, Y  +641.581, Z    +0.000, E1   -69.837, E3 +122091.049}
SPL {X  -160.000, Y  +657.932, Z    +0.000, E1   -69.833, E3 +122103.807}
SPL {X  -159.989, Y  +676.310, Z    +0.000, E1   -69.844, E3 +122118.115}
SPL {X  -158.945, Y  +692.747, Z    +0.000, E1   -69.717, E3 +122132.043}
SPL {X  -156.998, Y  +705.248, Z    +0.000, E1   -69.481, E3 +122143.830}
SPL {X  -153.152, Y  +720.707, Z    +0.000, E1   -69.072, E3 +122159.741}
SPL {X  -148.823, Y  +733.152, Z    +0.000, E1   -68.450, E3 +122173.900}
SPL {X  -145.304, Y  +741.384, Z    +0.000, E1   -67.989, E3 +122183.700}
SPL {X  -141.481, Y  +749.119, Z    +0.000, E1   -67.448, E3 +122193.325}
SPL {X  -137.717, Y  +755.849, Z    +0.000, E1   -66.896, E3 +122201.959}
SPL {X  -133.615, Y  +762.417, Z    +0.000, E1   -66.275, E3 +122210.574}
SPL {X  -128.952, Y  +769.117, Z    +0.000, E1   -65.522, E3 +122219.535}
SPL {X  -125.615, Y  +773.501, Z    +0.000, E1   -64.909, E3 +122225.472}
SPL {X   -93.482, Y  +804.250, Z    +0.000, E1   -52.853, E3 +122362.670}
ENDSPLINE

SPLINE
SPL {X  -137.039, Y  +756.986, Z    +0.000, E1   -45.206, E3 +122493.333}
SPL {X  -152.094, Y  +724.074, Z    +0.000, E1   -34.132, E3 +122509.280}
SPL {X  -158.930, Y  +692.872, Z    +0.000, E1   -16.505, E3 +122515.595}
SPL {X  -160.000, Y  +673.072, Z    +0.000, E1    -0.858, E3 +122516.906}
SPL {X  -160.000, Y  +670.505, Z    +0.000, E1    +2.991, E3 +122516.942}
SPL {X  -160.000, Y  +665.157, Z    +0.000, E1   +13.199, E3 +122517.172}
SPL {X  -160.000, Y  +657.552, Z    +0.000, E1   +28.428, E3 +122517.857}
SPL {X  -160.000, Y  +642.088, Z    +0.000, E1   +49.428, E3 +122520.847}
SPL {X  -160.000, Y  +582.331, Z    +0.000, E1   +67.139, E3 +122543.314}
SPL {X  -160.000, Y  +443.344, Z    +0.000, E1   +69.515, E3 +122627.800}
SPL {X  -160.000, Y  +423.295, Z    +0.000, E1   +69.546, E3 +122643.620}
SPL {X  -155.937, Y  +349.874, Z    +0.000, E1   +73.941, E3 +122651.691}
SPL {X  -155.646, Y  +348.628, Z    +0.000, E1   +73.073, E3 +122661.574}
SPL {X  -155.163, Y  +346.655, Z    +0.000, E1   +71.976, E3 +122673.561}
SPL {X  -154.105, Y  +342.669, Z    +0.000, E1   +70.814, E3 +122687.066}
SPL {X  -152.951, Y  +338.733, Z    +0.000, E1   +69.529, E3 +122700.910}
SPL {X  -150.673, Y  +331.871, Z    +0.000, E1   +68.778, E3 +122712.158}
SPL {X  -146.876, Y  +322.238, Z    +0.000, E1   +68.294, E3 +122723.339}
SPL {X  -142.952, Y  +313.834, Z    +0.000, E1   +67.744, E3 +122733.618}
SPL {X  -139.245, Y  +306.891, Z    +0.000, E1   +67.208, E3 +122742.402}
SPL {X  -135.108, Y  +299.992, Z    +0.000, E1   +66.599, E3 +122751.353}
SPL {X  -130.642, Y  +293.328, Z    +0.000, E1   +65.888, E3 +122760.205}
SPL {X  -126.461, Y  +287.682, Z    +0.000, E1   +65.179, E3 +122767.768}
SPL {X   -93.259, Y  +255.690, Z    +0.000, E1   +54.095, E3 +122883.150}
ENDSPLINE

SPLINE
SPL {X  -130.811, Y  +293.568, Z    +0.000, E1   +46.951, E3 +123027.010}
SPL {X  -151.580, Y  +334.479, Z    +0.000, E1   +34.520, E3 +123051.133}
SPL {X  -157.897, Y  +359.846, Z    +0.000, E1   +21.040, E3 +123057.091}
SPL {X  -159.671, Y  +375.443, Z    +0.000, E1   +10.084, E3 +123058.906}
SPL {X  -160.000, Y  +387.403, Z    +0.000, E1    +0.377, E3 +123059.382}
SPL {X  -160.000, Y  +391.807, Z    +0.000, E1    -7.102, E3 +123059.486}
SPL {X  -160.000, Y  +398.244, Z    +0.000, E1   -19.803, E3 +123059.920}
SPL {X  -160.000, Y  +410.795, Z    +0.000, E1   -41.112, E3 +123061.732}
SPL {X  -160.000, Y  +461.796, Z    +0.000, E1   -65.564, E3 +123078.375}
SPL {X  -160.000, Y  +623.854, Z    +0.000, E1   -69.845, E3 +123172.448}
SPL {X  -160.000, Y  +641.581, Z    +0.000, E1   -69.837, E3 +123186.287}
SPL {X  -160.000, Y  +657.932, Z    +0.000, E1   -69.833, E3 +123199.046}
SPL {X  -159.989, Y  +676.310, Z    +0.000, E1   -69.844, E3 +123213.354}
SPL {X  -158.945, Y  +692.747, Z    +0.000, E1   -69.717, E3 +123227.282}
SPL {X  -156.998, Y  +705.248, Z    +0.000, E1   -69.481, E3 +123239.069}
SPL {X  -153.152, Y  +720.707, Z    +0.000, E1   -69.072, E3 +123254.980}
SPL {X  -148.823, Y  +733.152, Z    +0.000, E1   -68.450, E3 +123269.139}
SPL {X  -145.304, Y  +741.384, Z    +0.000, E1   -67.989, E3 +123278.939}
SPL {X  -141.481, Y  +749.119, Z    +0.000, E1   -67.448, E3 +123288.564}
SPL {X  -137.717, Y  +755.849, Z    +0.000, E1   -66.896, E3 +123297.198}
SPL {X  -133.615, Y  +762.417, Z    +0.000, E1   -66.275, E3 +123305.812}
SPL {X  -128.952, Y  +769.117, Z    +0.000, E1   -65.522, E3 +123314.774}
SPL {X  -125.615, Y  +773.501, Z    +0.000, E1   -64.909, E3 +123320.711}
SPL {X   -93.482, Y  +804.250, Z    +0.000, E1   -52.853, E3 +123457.909}
ENDSPLINE

SPLINE
SPL {X  -137.039, Y  +756.986, Z    +0.000, E1   -45.206, E3 +123588.571}
SPL {X  -152.094, Y  +724.074, Z    +0.000, E1   -34.132, E3 +123604.518}
SPL {X  -158.930, Y  +692.872, Z    +0.000, E1   -16.505, E3 +123610.834}
SPL {X  -160.000, Y  +673.072, Z    +0.000, E1    -0.858, E3 +123612.145}
SPL {X  -160.000, Y  +670.505, Z    +0.000, E1    +2.991, E3 +123612.181}
SPL {X  -160.000, Y  +665.157, Z    +0.000, E1   +13.199, E3 +123612.411}
SPL {X  -160.000, Y  +657.552, Z    +0.000, E1   +28.428, E3 +123613.096}
SPL {X  -160.000, Y  +642.088, Z    +0.000, E1   +49.428, E3 +123616.086}
SPL {X  -160.000, Y  +582.331, Z    +0.000, E1   +67.139, E3 +123638.553}
SPL {X  -160.000, Y  +443.344, Z    +0.000, E1   +69.515, E3 +123723.039}
SPL {X  -160.000, Y  +423.295, Z    +0.000, E1   +69.546, E3 +123738.859}
SPL {X  -155.937, Y  +349.874, Z    +0.000, E1   +73.941, E3 +123746.930}
SPL {X  -155.646, Y  +348.628, Z    +0.000, E1   +73.073, E3 +123756.813}
SPL {X  -155.163, Y  +346.655, Z    +0.000, E1   +71.976, E3 +123768.800}
SPL {X  -154.105, Y  +342.669, Z    +0.000, E1   +70.814, E3 +123782.305}
SPL {X  -152.951, Y  +338.733, Z    +0.000, E1   +69.529, E3 +123796.149}
SPL {X  -150.673, Y  +331.871, Z    +0.000, E1   +68.778, E3 +123807.397}
SPL {X  -146.876, Y  +322.238, Z    +0.000, E1   +68.294, E3 +123818.577}
SPL {X  -142.952, Y  +313.834, Z    +0.000, E1   +67.744, E3 +123828.856}
SPL {X  -139.245, Y  +306.891, Z    +0.000, E1   +67.208, E3 +123837.640}
SPL {X  -135.108, Y  +299.992, Z    +0.000, E1   +66.599, E3 +123846.591}
SPL {X  -130.642, Y  +293.328, Z    +0.000, E1   +65.888, E3 +123855.444}
SPL {X  -126.461, Y  +287.682, Z    +0.000, E1   +65.179, E3 +123863.007}
SPL {X   -93.259, Y  +255.690, Z    +0.000, E1   +54.095, E3 +123978.388}
ENDSPLINE

SPLINE
SPL {X  -130.811, Y  +293.568, Z    +0.000, E1   +46.951, E3 +124122.249}
SPL {X  -151.580, Y  +334.479, Z    +0.000, E1   +34.520, E3 +124146.372}
SPL {X  -157.897, Y  +359.846, Z    +0.000, E1   +21.040, E3 +124152.329}
SPL {X  -159.671, Y  +375.443, Z    +0.000, E1   +10.084, E3 +124154.145}
SPL {X  -160.000, Y  +387.403, Z    +0.000, E1    +0.377, E3 +124154.620}
SPL {X  -160.000, Y  +391.807, Z    +0.000, E1    -7.102, E3 +124154.724}
SPL {X  -160.000, Y  +398.244, Z    +0.000, E1   -19.803, E3 +124155.158}
SPL {X  -160.000, Y  +410.795, Z    +0.000, E1   -41.112, E3 +124156.971}
SPL {X  -160.000, Y  +461.796, Z    +0.000, E1   -65.564, E3 +124173.614}
SPL {X  -160.000, Y  +623.854, Z    +0.000, E1   -69.845, E3 +124267.687}
SPL {X  -160.000, Y  +641.581, Z    +0.000, E1   -69.837, E3 +124281.526}
SPL {X  -160.000, Y  +657.932, Z    +0.000, E1   -69.833, E3 +124294.284}
SPL {X  -159.989, Y  +676.310, Z    +0.000, E1   -69.844, E3 +124308.592}
SPL {X  -158.945, Y  +692.747, Z    +0.000, E1   -69.717, E3 +124322.520}
SPL {X  -156.998, Y  +705.248, Z    +0.000, E1   -69.481, E3 +124334.307}
SPL {X  -153.152, Y  +720.707, Z    +0.000, E1   -69.072, E3 +124350.219}
SPL {X  -148.823, Y  +733.152, Z    +0.000, E1   -68.450, E3 +124364.378}
SPL {X  -145.304, Y  +741.384, Z    +0.000, E1   -67.989, E3 +124374.178}
SPL {X  -141.481, Y  +749.119, Z    +0.000, E1   -67.448, E3 +124383.802}
SPL {X  -137.717, Y  +755.849, Z    +0.000, E1   -66.896, E3 +124392.437}
SPL {X  -133.615, Y  +762.417, Z    +0.000, E1   -66.275, E3 +124401.051}
SPL {X  -128.952, Y  +769.117, Z    +0.000, E1   -65.522, E3 +124410.013}
SPL {X  -125.615, Y  +773.501, Z    +0.000, E1   -64.909, E3 +124415.950}
SPL {X   -93.482, Y  +804.250, Z    +0.000, E1   -52.853, E3 +124553.147}
ENDSPLINE

SPLINE
SPL {X  -137.039, Y  +756.986, Z    +0.000, E1   -45.206, E3 +124683.810}
SPL {X  -152.094, Y  +724.074, Z    +0.000, E1   -34.132, E3 +124699.757}
SPL {X  -158.930, Y  +692.872, Z    +0.000, E1   -16.505, E3 +124706.073}
SPL {X  -160.000, Y  +673.072, Z    +0.000, E1    -0.858, E3 +124707.383}
SPL {X  -160.000, Y  +670.505, Z    +0.000, E1    +2.991, E3 +124707.420}
SPL {X  -160.000, Y  +665.157, Z    +0.000, E1   +13.199, E3 +124707.649}
SPL {X  -160.000, Y  +657.552, Z    +0.000, E1   +28.428, E3 +124708.334}
SPL {X  -160.000, Y  +642.088, Z    +0.000, E1   +49.428, E3 +124711.324}
SPL {X  -160.000, Y  +582.331, Z    +0.000, E1   +67.139, E3 +124733.791}
SPL {X  -160.000, Y  +443.344, Z    +0.000, E1   +69.515, E3 +124818.278}
SPL {X  -160.000, Y  +423.295, Z    +0.000, E1   +69.546, E3 +124834.098}
SPL {X  -155.937, Y  +349.874, Z    +0.000, E1   +73.941, E3 +124842.168}
SPL {X  -155.646, Y  +348.628, Z    +0.000, E1   +73.073, E3 +124852.051}
SPL {X  -155.163, Y  +346.655, Z    +0.000, E1   +71.976, E3 +124864.039}
SPL {X  -154.105, Y  +342.669, Z    +0.000, E1   +70.814, E3 +124877.544}
SPL {X  -152.951, Y  +338.733, Z    +0.000, E1   +69.529, E3 +124891.387}
SPL {X  -150.673, Y  +331.871, Z    +0.000, E1   +68.778, E3 +124902.635}
SPL {X  -146.876, Y  +322.238, Z    +0.000, E1   +68.294, E3 +124913.816}
SPL {X  -142.952, Y  +313.834, Z    +0.000, E1   +67.744, E3 +124924.095}
SPL {X  -139.245, Y  +306.891, Z    +0.000, E1   +67.208, E3 +124932.879}
SPL {X  -135.108, Y  +299.992, Z    +0.000, E1   +66.599, E3 +124941.830}
SPL {X  -130.642, Y  +293.328, Z    +0.000, E1   +65.888, E3 +124950.682}
SPL {X  -126.461, Y  +287.682, Z    +0.000, E1   +65.179, E3 +124958.245}
SPL {X   -93.259, Y  +255.690, Z    +0.000, E1   +54.095, E3 +125073.627}
ENDSPLINE

SPLINE
SPL {X  -130.811, Y  +293.568, Z    +0.000, E1   +46.951, E3 +125217.488}
SPL {X  -151.580, Y  +334.479, Z    +0.000, E1   +34.520, E3 +125241.610}
SPL {X  -157.897, Y  +359.846, Z    +0.000, E1   +21.040, E3 +125247.568}
SPL {X  -159.671, Y  +375.443, Z    +0.000, E1   +10.084, E3 +125249.383}
SPL {X  -160.000, Y  +387.403, Z    +0.000, E1    +0.377, E3 +125249.859}
SPL {X  -160.000, Y  +391.807, Z    +0.000, E1    -7.102, E3 +125249.963}
SPL {X  -160.000, Y  +398.244, Z    +0.000, E1   -19.803, E3 +125250.397}
SPL {X  -160.000, Y  +410.795, Z    +0.000, E1   -41.112, E3 +125252.210}
SPL {X  -160.000, Y  +461.796, Z    +0.000, E1   -65.564, E3 +125268.853}
SPL {X  -160.000, Y  +623.854, Z    +0.000, E1   -69.845, E3 +125362.925}
SPL {X  -160.000, Y  +641.581, Z    +0.000, E1   -69.837, E3 +125376.765}
SPL {X  -160.000, Y  +657.932, Z    +0.000, E1   -69.833, E3 +125389.523}
SPL {X  -159.989, Y  +676.310, Z    +0.000, E1   -69.844, E3 +125403.831}
SPL {X  -158.945, Y  +692.747, Z    +0.000, E1   -69.717, E3 +125417.759}
SPL {X  -156.998, Y  +705.248, Z    +0.000, E1   -69.481, E3 +125429.546}
SPL {X  -153.152, Y  +720.707, Z    +0.000, E1   -69.072, E3 +125445.457}
SPL {X  -148.823, Y  +733.152, Z    +0.000, E1   -68.450, E3 +125459.616}
SPL {X  -145.304, Y  +741.384, Z    +0.000, E1   -67.989, E3 +125469.416}
SPL {X  -141.481, Y  +749.119, Z    +0.000, E1   -67.448, E3 +125479.041}
SPL {X  -137.717, Y  +755.849, Z    +0.000, E1   -66.896, E3 +125487.675}
SPL {X  -133.615, Y  +762.417, Z    +0.000, E1   -66.275, E3 +125496.290}
SPL {X  -128.952, Y  +769.117, Z    +0.000, E1   -65.522, E3 +125505.251}
SPL {X  -125.615, Y  +773.501, Z    +0.000, E1   -64.909, E3 +125511.188}
SPL {X   -93.482, Y  +804.250, Z    +0.000, E1   -52.853, E3 +125648.386}
ENDSPLINE

SPLINE
SPL {X  -137.039, Y  +756.986, Z    +0.000, E1   -45.206, E3 +125779.049}
SPL {X  -152.094, Y  +724.074, Z    +0.000, E1   -34.132, E3 +125794.996}
SPL {X  -158.930, Y  +692.872, Z    +0.000, E1   -16.505, E3 +125801.311}
SPL {X  -160.000, Y  +673.072, Z    +0.000, E1    -0.858, E3 +125802.622}
SPL {X  -160.000, Y  +670.505, Z    +0.000, E1    +2.991, E3 +125802.658}
SPL {X  -160.000, Y  +665.157, Z    +0.000, E1   +13.199, E3 +125802.888}
SPL {X  -160.000, Y  +657.552, Z    +0.000, E1   +28.428, E3 +125803.573}
SPL {X  -160.000, Y  +642.088, Z    +0.000, E1   +49.428, E3 +125806.563}
SPL {X  -160.000, Y  +582.331, Z    +0.000, E1   +67.139, E3 +125829.030}
SPL {X  -160.000, Y  +443.344, Z    +0.000, E1   +69.515, E3 +125913.516}
SPL {X  -160.000, Y  +423.295, Z    +0.000, E1   +69.546, E3 +125929.336}
SPL {X  -155.937, Y  +349.874, Z    +0.000, E1   +73.941, E3 +125937.407}
SPL {X  -155.646, Y  +348.628, Z    +0.000, E1   +73.073, E3 +125947.290}
SPL {X  -155.163, Y  +346.655, Z    +0.000, E1   +71.976, E3 +125959.277}
SPL {X  -154.105, Y  +342.669, Z    +0.000, E1   +70.814, E3 +125972.782}
SPL {X  -152.951, Y  +338.733, Z    +0.000, E1   +69.529, E3 +125986.626}
SPL {X  -150.673, Y  +331.871, Z    +0.000, E1   +68.778, E3 +125997.874}
SPL {X  -146.876, Y  +322.238, Z    +0.000, E1   +68.294, E3 +126009.055}
SPL {X  -142.952, Y  +313.834, Z    +0.000, E1   +67.744, E3 +126019.334}
SPL {X  -139.245, Y  +306.891, Z    +0.000, E1   +67.208, E3 +126028.118}
SPL {X  -135.108, Y  +299.992, Z    +0.000, E1   +66.599, E3 +126037.069}
SPL {X  -130.642, Y  +293.328, Z    +0.000, E1   +65.888, E3 +126045.921}
SPL {X  -126.461, Y  +287.682, Z    +0.000, E1   +65.179, E3 +126053.484}
SPL {X   -93.259, Y  +255.690, Z    +0.000, E1   +54.095, E3 +126168.866}
ENDSPLINE

SPLINE
SPL {X  -130.811, Y  +293.568, Z    +0.000, E1   +46.951, E3 +126312.726}
SPL {X  -151.580, Y  +334.479, Z    +0.000, E1   +34.520, E3 +126336.849}
SPL {X  -157.897, Y  +359.846, Z    +0.000, E1   +21.040, E3 +126342.807}
SPL {X  -159.671, Y  +375.443, Z    +0.000, E1   +10.084, E3 +126344.622}
SPL {X  -160.000, Y  +387.403, Z    +0.000, E1    +0.377, E3 +126345.098}
SPL {X  -160.000, Y  +391.807, Z    +0.000, E1    -7.102, E3 +126345.202}
SPL {X  -160.000, Y  +398.244, Z    +0.000, E1   -19.803, E3 +126345.636}
SPL {X  -160.000, Y  +410.795, Z    +0.000, E1   -41.112, E3 +126347.448}
SPL {X  -160.000, Y  +461.796, Z    +0.000, E1   -65.564, E3 +126364.091}
SPL {X  -160.000, Y  +623.854, Z    +0.000, E1   -69.845, E3 +126458.164}
SPL {X  -160.000, Y  +641.581, Z    +0.000, E1   -69.837, E3 +126472.003}
SPL {X  -160.000, Y  +657.932, Z    +0.000, E1   -69.833, E3 +126484.762}
SPL {X  -159.989, Y  +676.310, Z    +0.000, E1   -69.844, E3 +126499.070}
SPL {X  -158.945, Y  +692.747, Z    +0.000, E1   -69.717, E3 +126512.998}
SPL {X  -156.998, Y  +705.248, Z    +0.000, E1   -69.481, E3 +126524.785}
SPL {X  -153.152, Y  +720.707, Z    +0.000, E1   -69.072, E3 +126540.696}
SPL {X  -148.823, Y  +733.152, Z    +0.000, E1   -68.450, E3 +126554.855}
SPL {X  -145.304, Y  +741.384, Z    +0.000, E1   -67.989, E3 +126564.655}
SPL {X  -141.481, Y  +749.119, Z    +0.000, E1   -67.448, E3 +126574.280}
SPL {X  -137.717, Y  +755.849, Z    +0.000, E1   -66.896, E3 +126582.914}
SPL {X  -133.615, Y  +762.417, Z    +0.000, E1   -66.275, E3 +126591.528}
SPL {X  -128.952, Y  +769.117, Z    +0.000, E1   -65.522, E3 +126600.490}
SPL {X  -125.615, Y  +773.501, Z    +0.000, E1   -64.909, E3 +126606.427}
SPL {X   -93.482, Y  +804.250, Z    +0.000, E1   -52.853, E3 +126743.625}
ENDSPLINE

SPLINE
SPL {X  -137.039, Y  +756.986, Z    +0.000, E1   -45.206, E3 +126874.287}
SPL {X  -152.094, Y  +724.074, Z    +0.000, E1   -34.132, E3 +126890.234}
SPL {X  -158.930, Y  +692.872, Z    +0.000, E1   -16.505, E3 +126896.550}
SPL {X  -160.000, Y  +673.072, Z    +0.000, E1    -0.858, E3 +126897.861}
SPL {X  -160.000, Y  +670.505, Z    +0.000, E1    +2.991, E3 +126897.897}
SPL {X  -160.000, Y  +665.157, Z    +0.000, E1   +13.199, E3 +126898.127}
SPL {X  -160.000, Y  +657.552, Z    +0.000, E1   +28.428, E3 +126898.812}
SPL {X  -160.000, Y  +642.088, Z    +0.000, E1   +49.428, E3 +126901.802}
SPL {X  -160.000, Y  +582.331, Z    +0.000, E1   +67.139, E3 +126924.269}
SPL {X  -160.000, Y  +443.344, Z    +0.000, E1   +69.515, E3 +127008.755}
SPL {X  -160.000, Y  +423.295, Z    +0.000, E1   +69.546, E3 +127024.575}
SPL {X  -155.937, Y  +349.874, Z    +0.000, E1   +73.941, E3 +127032.646}
SPL {X  -155.646, Y  +348.628, Z    +0.000, E1   +73.073, E3 +127042.529}
SPL {X  -155.163, Y  +346.655, Z    +0.000, E1   +71.976, E3 +127054.516}
SPL {X  -154.105, Y  +342.669, Z    +0.000, E1   +70.814, E3 +127068.021}
SPL {X  -152.951, Y  +338.733, Z    +0.000, E1   +69.529, E3 +127081.865}
SPL {X  -150.673, Y  +331.871, Z    +0.000, E1   +68.778, E3 +127093.113}
SPL {X  -146.876, Y  +322.238, Z    +0.000, E1   +68.294, E3 +127104.293}
SPL {X  -142.952, Y  +313.834, Z    +0.000, E1   +67.744, E3 +127114.572}
SPL {X  -139.245, Y  +306.891, Z    +0.000, E1   +67.208, E3 +127123.356}
SPL {X  -135.108, Y  +299.992, Z    +0.000, E1   +66.599, E3 +127132.307}
SPL {X  -130.642, Y  +293.328, Z    +0.000, E1   +65.888, E3 +127141.160}
SPL {X  -126.461, Y  +287.682, Z    +0.000, E1   +65.179, E3 +127148.723}
SPL {X   -93.259, Y  +255.690, Z    +0.000, E1   +54.095, E3 +127264.104}
ENDSPLINE

SPLINE
SPL {X  -130.811, Y  +293.568, Z    +0.000, E1   +46.951, E3 +127407.965}
SPL {X  -151.580, Y  +334.479, Z    +0.000, E1   +34.520, E3 +127432.088}
SPL {X  -157.897, Y  +359.846, Z    +0.000, E1   +21.040, E3 +127438.045}
SPL {X  -159.671, Y  +375.443, Z    +0.000, E1   +10.084, E3 +127439.861}
SPL {X  -160.000, Y  +387.403, Z    +0.000, E1    +0.377, E3 +127440.336}
SPL {X  -160.000, Y  +391.807, Z    +0.000, E1    -7.102, E3 +127440.441}
SPL {X  -160.000, Y  +398.244, Z    +0.000, E1   -19.803, E3 +127440.874}
SPL {X  -160.000, Y  +410.795, Z    +0.000, E1   -41.112, E3 +127442.687}
SPL {X  -160.000, Y  +461.796, Z    +0.000, E1   -65.564, E3 +127459.330}
SPL {X  -160.000, Y  +623.854, Z    +0.000, E1   -69.845, E3 +127553.403}
SPL {X  -160.000, Y  +641.581, Z    +0.000, E1   -69.837, E3 +127567.242}
SPL {X  -160.000, Y  +657.932, Z    +0.000, E1   -69.833, E3 +127580.000}
SPL {X  -159.989, Y  +676.310, Z    +0.000, E1   -69.844, E3 +127594.308}
SPL {X  -158.945, Y  +692.747, Z    +0.000, E1   -69.717, E3 +127608.236}
SPL {X  -156.998, Y  +705.248, Z    +0.000, E1   -69.481, E3 +127620.023}
SPL {X  -153.152, Y  +720.707, Z    +0.000, E1   -69.072, E3 +127635.935}
SPL {X  -148.823, Y  +733.152, Z    +0.000, E1   -68.450, E3 +127650.094}
SPL {X  -145.304, Y  +741.384, Z    +0.000, E1   -67.989, E3 +127659.894}
SPL {X  -141.481, Y  +749.119, Z    +0.000, E1   -67.448, E3 +127669.518}
SPL {X  -137.717, Y  +755.849, Z    +0.000, E1   -66.896, E3 +127678.153}
SPL {X  -133.615, Y  +762.417, Z    +0.000, E1   -66.275, E3 +127686.767}
SPL {X  -128.952, Y  +769.117, Z    +0.000, E1   -65.522, E3 +127695.729}
SPL {X  -125.615, Y  +773.501, Z    +0.000, E1   -64.909, E3 +127701.666}
SPL {X   -93.482, Y  +804.250, Z    +0.000, E1   -52.853, E3 +127838.863}
ENDSPLINE

SPLINE
SPL {X  -137.039, Y  +756.986, Z    +0.000, E1   -45.206, E3 +127969.526}
SPL {X  -152.094, Y  +724.074, Z    +0.000, E1   -34.132, E3 +127985.473}
SPL {X  -158.930, Y  +692.872, Z    +0.000, E1   -16.505, E3 +127991.789}
SPL {X  -160.000, Y  +673.072, Z    +0.000, E1    -0.858, E3 +127993.099}
SPL {X  -160.000, Y  +670.505, Z    +0.000, E1    +2.991, E3 +127993.136}
SPL {X  -160.000, Y  +665.157, Z    +0.000, E1   +13.199, E3 +127993.365}
SPL {X  -160.000, Y  +657.552, Z    +0.000, E1   +28.428, E3 +127994.051}
SPL {X  -160.000, Y  +642.088, Z    +0.000, E1   +49.428, E3 +127997.040}
SPL {X  -160.000, Y  +582.331, Z    +0.000, E1   +67.139, E3 +128019.507}
SPL {X  -160.000, Y  +443.344, Z    +0.000, E1   +69.515, E3 +128103.994}
SPL {X  -160.000, Y  +423.295, Z    +0.000, E1   +69.546, E3 +128119.814}
SPL {X  -155.937, Y  +349.874, Z    +0.000, E1   +73.941, E3 +128127.884}
SPL {X  -155.646, Y  +348.628, Z    +0.000, E1   +73.073, E3 +128137.767}
SPL {X  -155.163, Y  +346.655, Z    +0.000, E1   +71.976, E3 +128149.755}
SPL {X  -154.105, Y  +342.669, Z    +0.000, E1   +70.814, E3 +128163.260}
SPL {X  -152.951, Y  +338.733, Z    +0.000, E1   +69.529, E3 +128177.103}
SPL {X  -150.673, Y  +331.871, Z    +0.000, E1   +68.778, E3 +128188.351}
SPL {X  -146.876, Y  +322.238, Z    +0.000, E1   +68.294, E3 +128199.532}
SPL {X  -142.952, Y  +313.834, Z    +0.000, E1   +67.744, E3 +128209.811}
SPL {X  -139.245, Y  +306.891, Z    +0.000, E1   +67.208, E3 +128218.595}
SPL {X  -135.108, Y  +299.992, Z    +0.000, E1   +66.599, E3 +128227.546}
SPL {X  -130.642, Y  +293.328, Z    +0.000, E1   +65.888, E3 +128236.398}
SPL {X  -126.461, Y  +287.682, Z    +0.000, E1   +65.179, E3 +128243.961}
SPL {X   -93.259, Y  +255.690, Z    +0.000, E1   +54.095, E3 +128359.343}
ENDSPLINE

SPLINE
SPL {X  -130.811, Y  +293.568, Z    +0.000, E1   +46.951, E3 +128503.204}
SPL {X  -151.580, Y  +334.479, Z    +0.000, E1   +34.520, E3 +128527.326}
SPL {X  -157.897, Y  +359.846, Z    +0.000, E1   +21.040, E3 +128533.284}
SPL {X  -159.671, Y  +375.443, Z    +0.000, E1   +10.084, E3 +128535.099}
SPL {X  -160.000, Y  +387.403, Z    +0.000, E1    +0.377, E3 +128535.575}
SPL {X  -160.000, Y  +391.807, Z    +0.000, E1    -7.102, E3 +128535.679}
SPL {X  -160.000, Y  +398.244, Z    +0.000, E1   -19.803, E3 +128536.113}
SPL {X  -160.000, Y  +410.795, Z    +0.000, E1   -41.112, E3 +128537.926}
SPL {X  -160.000, Y  +461.796, Z    +0.000, E1   -65.564, E3 +128554.569}
SPL {X  -160.000, Y  +623.854, Z    +0.000, E1   -69.845, E3 +128648.641}
SPL {X  -160.000, Y  +641.581, Z    +0.000, E1   -69.837, E3 +128662.481}
SPL {X  -160.000, Y  +657.932, Z    +0.000, E1   -69.833, E3 +128675.239}
SPL {X  -159.989, Y  +676.310, Z    +0.000, E1   -69.844, E3 +128689.547}
SPL {X  -158.945, Y  +692.747, Z    +0.000, E1   -69.717, E3 +128703.475}
SPL {X  -156.998, Y  +705.248, Z    +0.000, E1   -69.481, E3 +128715.262}
SPL {X  -153.152, Y  +720.707, Z    +0.000, E1   -69.072, E3 +128731.173}
SPL {X  -148.823, Y  +733.152, Z    +0.000, E1   -68.450, E3 +128745.332}
SPL {X  -145.304, Y  +741.384, Z    +0.000, E1   -67.989, E3 +128755.132}
SPL {X  -141.481, Y  +749.119, Z    +0.000, E1   -67.448, E3 +128764.757}
SPL {X  -137.717, Y  +755.849, Z    +0.000, E1   -66.896, E3 +128773.391}
SPL {X  -133.615, Y  +762.417, Z    +0.000, E1   -66.275, E3 +128782.006}
SPL {X  -128.952, Y  +769.117, Z    +0.000, E1   -65.522, E3 +128790.968}
SPL {X  -125.615, Y  +773.501, Z    +0.000, E1   -64.909, E3 +128796.904}
SPL {X   -93.482, Y  +804.250, Z    +0.000, E1   -52.853, E3 +128934.102}
ENDSPLINE

SPLINE
SPL {X  -137.039, Y  +756.986, Z    +0.000, E1   -45.206, E3 +129064.765}
SPL {X  -152.094, Y  +724.074, Z    +0.000, E1   -34.132, E3 +129080.712}
SPL {X  -158.930, Y  +692.872, Z    +0.000, E1   -16.505, E3 +129087.027}
SPL {X  -160.000, Y  +673.072, Z    +0.000, E1    -0.858, E3 +129088.338}
SPL {X  -160.000, Y  +670.505, Z    +0.000, E1    +2.991, E3 +129088.374}
SPL {X  -160.000, Y  +665.157, Z    +0.000, E1   +13.199, E3 +129088.604}
SPL {X  -160.000, Y  +657.552, Z    +0.000, E1   +28.428, E3 +129089.289}
SPL {X  -160.000, Y  +642.088, Z    +0.000, E1   +49.428, E3 +129092.279}
SPL {X  -160.000, Y  +582.331, Z    +0.000, E1   +67.139, E3 +129114.746}
SPL {X  -160.000, Y  +443.344, Z    +0.000, E1   +69.515, E3 +129199.232}
SPL {X  -160.000, Y  +423.295, Z    +0.000, E1   +69.546, E3 +129215.052}
SPL {X  -155.937, Y  +349.874, Z    +0.000, E1   +73.941, E3 +129223.123}
SPL {X  -155.646, Y  +348.628, Z    +0.000, E1   +73.073, E3 +129233.006}
SPL {X  -155.163, Y  +346.655, Z    +0.000, E1   +71.976, E3 +129244.993}
SPL {X  -154.105, Y  +342.669, Z    +0.000, E1   +70.814, E3 +129258.498}
SPL {X  -152.951, Y  +338.733, Z    +0.000, E1   +69.529, E3 +129272.342}
SPL {X  -150.673, Y  +331.871, Z    +0.000, E1   +68.778, E3 +129283.590}
SPL {X  -146.876, Y  +322.238, Z    +0.000, E1   +68.294, E3 +129294.771}
SPL {X  -142.952, Y  +313.834, Z    +0.000, E1   +67.744, E3 +129305.050}
SPL {X  -139.245, Y  +306.891, Z    +0.000, E1   +67.208, E3 +129313.834}
SPL {X  -135.108, Y  +299.992, Z    +0.000, E1   +66.599, E3 +129322.785}
SPL {X  -130.642, Y  +293.328, Z    +0.000, E1   +65.888, E3 +129331.637}
SPL {X  -126.461, Y  +287.682, Z    +0.000, E1   +65.179, E3 +129339.200}
SPL {X   -93.259, Y  +255.690, Z    +0.000, E1   +54.095, E3 +129454.582}
ENDSPLINE

SPLINE
SPL {X  -130.811, Y  +293.568, Z    +0.000, E1   +46.951, E3 +129598.442}
SPL {X  -151.580, Y  +334.479, Z    +0.000, E1   +34.520, E3 +129622.565}
SPL {X  -157.897, Y  +359.846, Z    +0.000, E1   +21.040, E3 +129628.523}
SPL {X  -159.671, Y  +375.443, Z    +0.000, E1   +10.084, E3 +129630.338}
SPL {X  -160.000, Y  +387.403, Z    +0.000, E1    +0.377, E3 +129630.814}
SPL {X  -160.000, Y  +391.807, Z    +0.000, E1    -7.102, E3 +129630.918}
SPL {X  -160.000, Y  +398.244, Z    +0.000, E1   -19.803, E3 +129631.352}
SPL {X  -160.000, Y  +410.795, Z    +0.000, E1   -41.112, E3 +129633.164}
SPL {X  -160.000, Y  +461.796, Z    +0.000, E1   -65.564, E3 +129649.807}
SPL {X  -160.000, Y  +623.854, Z    +0.000, E1   -69.845, E3 +129743.880}
SPL {X  -160.000, Y  +641.581, Z    +0.000, E1   -69.837, E3 +129757.719}
SPL {X  -160.000, Y  +657.932, Z    +0.000, E1   -69.833, E3 +129770.478}
SPL {X  -159.989, Y  +676.310, Z    +0.000, E1   -69.844, E3 +129784.786}
SPL {X  -158.945, Y  +692.747, Z    +0.000, E1   -69.717, E3 +129798.714}
SPL {X  -156.998, Y  +705.248, Z    +0.000, E1   -69.481, E3 +129810.501}
SPL {X  -153.152, Y  +720.707, Z    +0.000, E1   -69.072, E3 +129826.412}
SPL {X  -148.823, Y  +733.152, Z    +0.000, E1   -68.450, E3 +129840.571}
SPL {X  -145.304, Y  +741.384, Z    +0.000, E1   -67.989, E3 +129850.371}
SPL {X  -141.481, Y  +749.119, Z    +0.000, E1   -67.448, E3 +129859.996}
SPL {X  -137.717, Y  +755.849, Z    +0.000, E1   -66.896, E3 +129868.630}
SPL {X  -133.615, Y  +762.417, Z    +0.000, E1   -66.275, E3 +129877.244}
SPL {X  -128.952, Y  +769.117, Z    +0.000, E1   -65.522, E3 +129886.206}
SPL {X  -125.615, Y  +773.501, Z    +0.000, E1   -64.909, E3 +129892.143}
SPL {X   -93.482, Y  +804.250, Z    +0.000, E1   -52.853, E3 +130029.341}
ENDSPLINE

SPLINE
SPL {X  -137.039, Y  +756.986, Z    +0.000, E1   -45.206, E3 +130160.003}
SPL {X  -152.094, Y  +724.074, Z    +0.000, E1   -34.132, E3 +130175.950}
SPL {X  -158.930, Y  +692.872, Z    +0.000, E1   -16.505, E3 +130182.266}
SPL {X  -160.000, Y  +673.072, Z    +0.000, E1    -0.858, E3 +130183.577}
SPL {X  -160.000, Y  +670.505, Z    +0.000, E1    +2.991, E3 +130183.613}
SPL {X  -160.000, Y  +665.157, Z    +0.000, E1   +13.199, E3 +130183.843}
SPL {X  -160.000, Y  +657.552, Z    +0.000, E1   +28.428, E3 +130184.528}
SPL {X  -160.000, Y  +642.088, Z    +0.000, E1   +49.428, E3 +130187.518}
SPL {X  -160.000, Y  +582.331, Z    +0.000, E1   +67.139, E3 +130209.985}
SPL {X  -160.000, Y  +443.344, Z    +0.000, E1   +69.515, E3 +130294.471}
SPL {X  -160.000, Y  +423.295, Z    +0.000, E1   +69.546, E3 +130310.291}
SPL {X  -155.937, Y  +349.874, Z    +0.000, E1   +73.941, E3 +130318.362}
SPL {X  -155.646, Y  +348.628, Z    +0.000, E1   +73.073, E3 +130328.245}
SPL {X  -155.163, Y  +346.655, Z    +0.000, E1   +71.976, E3 +130340.232}
SPL {X  -154.105, Y  +342.669, Z    +0.000, E1   +70.814, E3 +130353.737}
SPL {X  -152.951, Y  +338.733, Z    +0.000, E1   +69.529, E3 +130367.581}
SPL {X  -150.673, Y  +331.871, Z    +0.000, E1   +68.778, E3 +130378.829}
SPL {X  -146.876, Y  +322.238, Z    +0.000, E1   +68.294, E3 +130390.010}
SPL {X  -142.952, Y  +313.834, Z    +0.000, E1   +67.744, E3 +130400.288}
SPL {X  -139.245, Y  +306.891, Z    +0.000, E1   +67.208, E3 +130409.072}
SPL {X  -135.108, Y  +299.992, Z    +0.000, E1   +66.599, E3 +130418.024}
SPL {X  -130.642, Y  +293.328, Z    +0.000, E1   +65.888, E3 +130426.876}
SPL {X  -126.461, Y  +287.682, Z    +0.000, E1   +65.179, E3 +130434.439}
SPL {X   -93.259, Y  +255.690, Z    +0.000, E1   +54.095, E3 +130549.820}
ENDSPLINE

SPLINE
SPL {X  -130.811, Y  +293.568, Z    +0.000, E1   +46.951, E3 +130693.681}
SPL {X  -151.580, Y  +334.479, Z    +0.000, E1   +34.520, E3 +130717.804}
SPL {X  -157.897, Y  +359.846, Z    +0.000, E1   +21.040, E3 +130723.761}
SPL {X  -159.671, Y  +375.443, Z    +0.000, E1   +10.084, E3 +130725.577}
SPL {X  -160.000, Y  +387.403, Z    +0.000, E1    +0.377, E3 +130726.052}
SPL {X  -160.000, Y  +391.807, Z    +0.000, E1    -7.102, E3 +130726.157}
SPL {X  -160.000, Y  +398.244, Z    +0.000, E1   -19.803, E3 +130726.590}
SPL {X  -160.000, Y  +410.795, Z    +0.000, E1   -41.112, E3 +130728.403}
SPL {X  -160.000, Y  +461.796, Z    +0.000, E1   -65.564, E3 +130745.046}
SPL {X  -160.000, Y  +623.854, Z    +0.000, E1   -69.845, E3 +130839.119}
SPL {X  -160.000, Y  +641.581, Z    +0.000, E1   -69.837, E3 +130852.958}
SPL {X  -160.000, Y  +657.932, Z    +0.000, E1   -69.833, E3 +130865.716}
SPL {X  -159.989, Y  +676.310, Z    +0.000, E1   -69.844, E3 +130880.024}
SPL {X  -158.945, Y  +692.747, Z    +0.000, E1   -69.717, E3 +130893.952}
SPL {X  -156.998, Y  +705.248, Z    +0.000, E1   -69.481, E3 +130905.739}
SPL {X  -153.152, Y  +720.707, Z    +0.000, E1   -69.072, E3 +130921.651}
SPL {X  -148.823, Y  +733.152, Z    +0.000, E1   -68.450, E3 +130935.810}
SPL {X  -145.304, Y  +741.384, Z    +0.000, E1   -67.989, E3 +130945.610}
SPL {X  -141.481, Y  +749.119, Z    +0.000, E1   -67.448, E3 +130955.234}
SPL {X  -137.717, Y  +755.849, Z    +0.000, E1   -66.896, E3 +130963.869}
SPL {X  -133.615, Y  +762.417, Z    +0.000, E1   -66.275, E3 +130972.483}
SPL {X  -128.952, Y  +769.117, Z    +0.000, E1   -65.522, E3 +130981.445}
SPL {X  -125.615, Y  +773.501, Z    +0.000, E1   -64.909, E3 +130987.382}
SPL {X   -93.482, Y  +804.250, Z    +0.000, E1   -52.853, E3 +131124.579}
ENDSPLINE

SPLINE
SPL {X  -137.039, Y  +756.986, Z    +0.000, E1   -45.206, E3 +131255.242}
SPL {X  -152.094, Y  +724.074, Z    +0.000, E1   -34.132, E3 +131271.189}
SPL {X  -158.930, Y  +692.872, Z    +0.000, E1   -16.505, E3 +131277.505}
SPL {X  -160.000, Y  +673.072, Z    +0.000, E1    -0.858, E3 +131278.815}
SPL {X  -160.000, Y  +670.505, Z    +0.000, E1    +2.991, E3 +131278.852}
SPL {X  -160.000, Y  +665.157, Z    +0.000, E1   +13.199, E3 +131279.081}
SPL {X  -160.000, Y  +657.552, Z    +0.000, E1   +28.428, E3 +131279.767}
SPL {X  -160.000, Y  +642.088, Z    +0.000, E1   +49.428, E3 +131282.756}
SPL {X  -160.000, Y  +582.331, Z    +0.000, E1   +67.139, E3 +131305.223}
SPL {X  -160.000, Y  +443.344, Z    +0.000, E1   +69.515, E3 +131389.710}
SPL {X  -160.000, Y  +423.295, Z    +0.000, E1   +69.546, E3 +131405.530}
SPL {X  -155.937, Y  +349.874, Z    +0.000, E1   +73.941, E3 +131413.600}
SPL {X  -155.646, Y  +348.628, Z    +0.000, E1   +73.073, E3 +131423.483}
SPL {X  -155.163, Y  +346.655, Z    +0.000, E1   +71.976, E3 +131435.471}
SPL {X  -154.105, Y  +342.669, Z    +0.000, E1   +70.814, E3 +131448.976}
SPL {X  -152.951, Y  +338.733, Z    +0.000, E1   +69.529, E3 +131462.819}
SPL {X  -150.673, Y  +331.871, Z    +0.000, E1   +68.778, E3 +131474.067}
SPL {X  -146.876, Y  +322.238, Z    +0.000, E1   +68.294, E3 +131485.248}
SPL {X  -142.952, Y  +313.834, Z    +0.000, E1   +67.744, E3 +131495.527}
SPL {X  -139.245, Y  +306.891, Z    +0.000, E1   +67.208, E3 +131504.311}
SPL {X  -135.108, Y  +299.992, Z    +0.000, E1   +66.599, E3 +131513.262}
SPL {X  -130.642, Y  +293.328, Z    +0.000, E1   +65.888, E3 +131522.114}
SPL {X  -126.461, Y  +287.682, Z    +0.000, E1   +65.179, E3 +131529.677}
SPL {X   -93.259, Y  +255.690, Z    +0.000, E1   +54.095, E3 +131645.059}
ENDSPLINE

SPLINE
SPL {X  -130.811, Y  +293.568, Z    +0.000, E1   +46.951, E3 +131788.920}
SPL {X  -151.580, Y  +334.479, Z    +0.000, E1   +34.520, E3 +131813.042}
SPL {X  -157.897, Y  +359.846, Z    +0.000, E1   +21.040, E3 +131819.000}
SPL {X  -159.671, Y  +375.443, Z    +0.000, E1   +10.084, E3 +131820.815}
SPL {X  -160.000, Y  +387.403, Z    +0.000, E1    +0.377, E3 +131821.291}
SPL {X  -160.000, Y  +391.807, Z    +0.000, E1    -7.102, E3 +131821.395}
SPL {X  -160.000, Y  +398.244, Z    +0.000, E1   -19.803, E3 +131821.829}
SPL {X  -160.000, Y  +410.795, Z    +0.000, E1   -41.112, E3 +131823.642}
SPL {X  -160.000, Y  +461.796, Z    +0.000, E1   -65.564, E3 +131840.285}
SPL {X  -160.000, Y  +623.854, Z    +0.000, E1   -69.845, E3 +131934.357}
SPL {X  -160.000, Y  +641.581, Z    +0.000, E1   -69.837, E3 +131948.197}
SPL {X  -160.000, Y  +657.932, Z    +0.000, E1   -69.833, E3 +131960.955}
SPL {X  -159.989, Y  +676.310, Z    +0.000, E1   -69.844, E3 +131975.263}
SPL {X  -158.945, Y  +692.747, Z    +0.000, E1   -69.717, E3 +131989.191}
SPL {X  -156.998, Y  +705.248, Z    +0.000, E1   -69.481, E3 +132000.978}
SPL {X  -153.152, Y  +720.707, Z    +0.000, E1   -69.072, E3 +132016.890}
SPL {X  -148.823, Y  +733.152, Z    +0.000, E1   -68.450, E3 +132031.048}
SPL {X  -145.304, Y  +741.384, Z    +0.000, E1   -67.989, E3 +132040.848}
SPL {X  -141.481, Y  +749.119, Z    +0.000, E1   -67.448, E3 +132050.473}
SPL {X  -137.717, Y  +755.849, Z    +0.000, E1   -66.896, E3 +132059.107}
SPL {X  -133.615, Y  +762.417, Z    +0.000, E1   -66.275, E3 +132067.722}
SPL {X  -128.952, Y  +769.117, Z    +0.000, E1   -65.522, E3 +132076.684}
SPL {X  -125.615, Y  +773.501, Z    +0.000, E1   -64.909, E3 +132082.620}
SPL {X   -93.482, Y  +804.250, Z    +0.000, E1   -52.853, E3 +132219.818}
ENDSPLINE

SPLINE
SPL {X  -137.039, Y  +756.986, Z    +0.000, E1   -45.206, E3 +132350.481}
SPL {X  -152.094, Y  +724.074, Z    +0.000, E1   -34.132, E3 +132366.428}
SPL {X  -158.930, Y  +692.872, Z    +0.000, E1   -16.505, E3 +132372.744}
SPL {X  -160.000, Y  +673.072, Z    +0.000, E1    -0.858, E3 +132374.054}
SPL {X  -160.000, Y  +670.505, Z    +0.000, E1    +2.991, E3 +132374.090}
SPL {X  -160.000, Y  +665.157, Z    +0.000, E1   +13.199, E3 +132374.320}
SPL {X  -160.000, Y  +657.552, Z    +0.000, E1   +28.428, E3 +132375.005}
SPL {X  -160.000, Y  +642.088, Z    +0.000, E1   +49.428, E3 +132377.995}
SPL {X  -160.000, Y  +582.331, Z    +0.000, E1   +67.139, E3 +132400.462}
SPL {X  -160.000, Y  +443.344, Z    +0.000, E1   +69.515, E3 +132484.948}
SPL {X  -160.000, Y  +423.295, Z    +0.000, E1   +69.546, E3 +132500.768}
SPL {X  -155.937, Y  +349.874, Z    +0.000, E1   +73.941, E3 +132508.839}
SPL {X  -155.646, Y  +348.628, Z    +0.000, E1   +73.073, E3 +132518.722}
SPL {X  -155.163, Y  +346.655, Z    +0.000, E1   +71.976, E3 +132530.709}
SPL {X  -154.105, Y  +342.669, Z    +0.000, E1   +70.814, E3 +132544.214}
SPL {X  -152.951, Y  +338.733, Z    +0.000, E1   +69.529, E3 +132558.058}
SPL {X  -150.673, Y  +331.871, Z    +0.000, E1   +68.778, E3 +132569.306}
SPL {X  -146.876, Y  +322.238, Z    +0.000, E1   +68.294, E3 +132580.487}
SPL {X  -142.952, Y  +313.834, Z    +0.000, E1   +67.744, E3 +132590.766}
SPL {X  -139.245, Y  +306.891, Z    +0.000, E1   +67.208, E3 +132599.550}
SPL {X  -135.108, Y  +299.992, Z    +0.000, E1   +66.599, E3 +132608.501}
SPL {X  -130.642, Y  +293.328, Z    +0.000, E1   +65.888, E3 +132617.353}
SPL {X  -126.461, Y  +287.682, Z    +0.000, E1   +65.179, E3 +132624.916}
SPL {X   -93.259, Y  +255.690, Z    +0.000, E1   +54.095, E3 +132740.298}
ENDSPLINE

SPLINE
SPL {X  -130.811, Y  +293.568, Z    +0.000, E1   +46.951, E3 +132884.158}
SPL {X  -151.580, Y  +334.479, Z    +0.000, E1   +34.520, E3 +132908.281}
SPL {X  -157.897, Y  +359.846, Z    +0.000, E1   +21.040, E3 +132914.239}
SPL {X  -159.671, Y  +375.443, Z    +0.000, E1   +10.084, E3 +132916.054}
SPL {X  -160.000, Y  +387.403, Z    +0.000, E1    +0.377, E3 +132916.530}
SPL {X  -160.000, Y  +391.807, Z    +0.000, E1    -7.102, E3 +132916.634}
SPL {X  -160.000, Y  +398.244, Z    +0.000, E1   -19.803, E3 +132917.068}
SPL {X  -160.000, Y  +410.795, Z    +0.000, E1   -41.112, E3 +132918.881}
SPL {X  -160.000, Y  +461.796, Z    +0.000, E1   -65.564, E3 +132935.523}
SPL {X  -160.000, Y  +623.854, Z    +0.000, E1   -69.845, E3 +133029.596}
SPL {X  -160.000, Y  +641.581, Z    +0.000, E1   -69.837, E3 +133043.435}
SPL {X  -160.000, Y  +657.932, Z    +0.000, E1   -69.833, E3 +133056.194}
SPL {X  -159.989, Y  +676.310, Z    +0.000, E1   -69.844, E3 +133070.502}
SPL {X  -158.945, Y  +692.747, Z    +0.000, E1   -69.717, E3 +133084.430}
SPL {X  -156.998, Y  +705.248, Z    +0.000, E1   -69.481, E3 +133096.217}
SPL {X  -153.152, Y  +720.707, Z    +0.000, E1   -69.072, E3 +133112.128}
SPL {X  -148.823, Y  +733.152, Z    +0.000, E1   -68.450, E3 +133126.287}
SPL {X  -145.304, Y  +741.384, Z    +0.000, E1   -67.989, E3 +133136.087}
SPL {X  -141.481, Y  +749.119, Z    +0.000, E1   -67.448, E3 +133145.712}
SPL {X  -137.717, Y  +755.849, Z    +0.000, E1   -66.896, E3 +133154.346}
SPL {X  -133.615, Y  +762.417, Z    +0.000, E1   -66.275, E3 +133162.961}
SPL {X  -128.952, Y  +769.117, Z    +0.000, E1   -65.522, E3 +133171.922}
SPL {X  -125.615, Y  +773.501, Z    +0.000, E1   -64.909, E3 +133177.859}
SPL {X   -93.482, Y  +804.250, Z    +0.000, E1   -52.853, E3 +133315.057}
ENDSPLINE

SPLINE
SPL {X  -137.039, Y  +756.986, Z    +0.000, E1   -45.206, E3 +133445.720}
SPL {X  -152.094, Y  +724.074, Z    +0.000, E1   -34.132, E3 +133461.666}
SPL {X  -158.930, Y  +692.872, Z    +0.000, E1   -16.505, E3 +133467.982}
SPL {X  -160.000, Y  +673.072, Z    +0.000, E1    -0.858, E3 +133469.293}
SPL {X  -160.000, Y  +670.505, Z    +0.000, E1    +2.991, E3 +133469.329}
SPL {X  -160.000, Y  +665.157, Z    +0.000, E1   +13.199, E3 +133469.559}
SPL {X  -160.000, Y  +657.552, Z    +0.000, E1   +28.428, E3 +133470.244}
SPL {X  -160.000, Y  +642.088, Z    +0.000, E1   +49.428, E3 +133473.234}
SPL {X  -160.000, Y  +582.331, Z    +0.000, E1   +67.139, E3 +133495.701}
SPL {X  -160.000, Y  +443.344, Z    +0.000, E1   +69.515, E3 +133580.187}
SPL {X  -160.000, Y  +423.295, Z    +0.000, E1   +69.546, E3 +133596.007}
SPL {X  -155.937, Y  +349.874, Z    +0.000, E1   +73.941, E3 +133604.078}
SPL {X  -155.646, Y  +348.628, Z    +0.000, E1   +73.073, E3 +133613.961}
SPL {X  -155.163, Y  +346.655, Z    +0.000, E1   +71.976, E3 +133625.948}
SPL {X  -154.105, Y  +342.669, Z    +0.000, E1   +70.814, E3 +133639.453}
SPL {X  -152.951, Y  +338.733, Z    +0.000, E1   +69.529, E3 +133653.297}
SPL {X  -150.673, Y  +331.871, Z    +0.000, E1   +68.778, E3 +133664.545}
SPL {X  -146.876, Y  +322.238, Z    +0.000, E1   +68.294, E3 +133675.726}
SPL {X  -142.952, Y  +313.834, Z    +0.000, E1   +67.744, E3 +133686.004}
SPL {X  -139.245, Y  +306.891, Z    +0.000, E1   +67.208, E3 +133694.788}
SPL {X  -135.108, Y  +299.992, Z    +0.000, E1   +66.599, E3 +133703.740}
SPL {X  -130.642, Y  +293.328, Z    +0.000, E1   +65.888, E3 +133712.592}
SPL {X  -126.461, Y  +287.682, Z    +0.000, E1   +65.179, E3 +133720.155}
SPL {X   -93.259, Y  +255.690, Z    +0.000, E1   +54.095, E3 +133835.537}
ENDSPLINE

SPLINE
SPL {X  -130.811, Y  +293.568, Z    +0.000, E1   +46.951, E3 +133979.397}
SPL {X  -151.580, Y  +334.479, Z    +0.000, E1   +34.520, E3 +134003.520}
SPL {X  -157.897, Y  +359.846, Z    +0.000, E1   +21.040, E3 +134009.478}
SPL {X  -159.671, Y  +375.443, Z    +0.000, E1   +10.084, E3 +134011.293}
SPL {X  -160.000, Y  +387.403, Z    +0.000, E1    +0.377, E3 +134011.768}
SPL {X  -160.000, Y  +391.807, Z    +0.000, E1    -7.102, E3 +134011.873}
SPL {X  -160.000, Y  +398.244, Z    +0.000, E1   -19.803, E3 +134012.306}
SPL {X  -160.000, Y  +410.795, Z    +0.000, E1   -41.112, E3 +134014.119}
SPL {X  -160.000, Y  +461.796, Z    +0.000, E1   -65.564, E3 +134030.762}
SPL {X  -160.000, Y  +623.854, Z    +0.000, E1   -69.845, E3 +134124.835}
SPL {X  -160.000, Y  +641.581, Z    +0.000, E1   -69.837, E3 +134138.674}
SPL {X  -160.000, Y  +657.932, Z    +0.000, E1   -69.833, E3 +134151.432}
SPL {X  -159.989, Y  +676.310, Z    +0.000, E1   -69.844, E3 +134165.740}
SPL {X  -158.945, Y  +692.747, Z    +0.000, E1   -69.717, E3 +134179.668}
SPL {X  -156.998, Y  +705.248, Z    +0.000, E1   -69.481, E3 +134191.455}
SPL {X  -153.152, Y  +720.707, Z    +0.000, E1   -69.072, E3 +134207.367}
SPL {X  -148.823, Y  +733.152, Z    +0.000, E1   -68.450, E3 +134221.526}
SPL {X  -145.304, Y  +741.384, Z    +0.000, E1   -67.989, E3 +134231.326}
SPL {X  -141.481, Y  +749.119, Z    +0.000, E1   -67.448, E3 +134240.950}
SPL {X  -137.717, Y  +755.849, Z    +0.000, E1   -66.896, E3 +134249.585}
SPL {X  -133.615, Y  +762.417, Z    +0.000, E1   -66.275, E3 +134258.199}
SPL {X  -128.952, Y  +769.117, Z    +0.000, E1   -65.522, E3 +134267.161}
SPL {X  -125.615, Y  +773.501, Z    +0.000, E1   -64.909, E3 +134273.098}
SPL {X   -93.482, Y  +804.250, Z    +0.000, E1   -52.853, E3 +134410.295}
ENDSPLINE

SPLINE
SPL {X  -137.039, Y  +756.986, Z    +0.000, E1   -45.206, E3 +134540.958}
SPL {X  -152.094, Y  +724.074, Z    +0.000, E1   -34.132, E3 +134556.905}
SPL {X  -158.930, Y  +692.872, Z    +0.000, E1   -16.505, E3 +134563.221}
SPL {X  -160.000, Y  +673.072, Z    +0.000, E1    -0.858, E3 +134564.531}
SPL {X  -160.000, Y  +670.505, Z    +0.000, E1    +2.991, E3 +134564.568}
SPL {X  -160.000, Y  +665.157, Z    +0.000, E1   +13.199, E3 +134564.797}
SPL {X  -160.000, Y  +657.552, Z    +0.000, E1   +28.428, E3 +134565.483}
SPL {X  -160.000, Y  +642.088, Z    +0.000, E1   +49.428, E3 +134568.473}
SPL {X  -160.000, Y  +582.331, Z    +0.000, E1   +67.139, E3 +134590.939}
SPL {X  -160.000, Y  +443.344, Z    +0.000, E1   +69.515, E3 +134675.426}
SPL {X  -160.000, Y  +423.295, Z    +0.000, E1   +69.546, E3 +134691.246}
SPL {X  -155.937, Y  +349.874, Z    +0.000, E1   +73.941, E3 +134699.316}
SPL {X  -155.646, Y  +348.628, Z    +0.000, E1   +73.073, E3 +134709.199}
SPL {X  -155.163, Y  +346.655, Z    +0.000, E1   +71.976, E3 +134721.187}
SPL {X  -154.105, Y  +342.669, Z    +0.000, E1   +70.814, E3 +134734.692}
SPL {X  -152.951, Y  +338.733, Z    +0.000, E1   +69.529, E3 +134748.535}
SPL {X  -150.673, Y  +331.871, Z    +0.000, E1   +68.778, E3 +134759.783}
SPL {X  -146.876, Y  +322.238, Z    +0.000, E1   +68.294, E3 +134770.964}
SPL {X  -142.952, Y  +313.834, Z    +0.000, E1   +67.744, E3 +134781.243}
SPL {X  -139.245, Y  +306.891, Z    +0.000, E1   +67.208, E3 +134790.027}
SPL {X  -135.108, Y  +299.992, Z    +0.000, E1   +66.599, E3 +134798.978}
SPL {X  -130.642, Y  +293.328, Z    +0.000, E1   +65.888, E3 +134807.830}
SPL {X  -126.461, Y  +287.682, Z    +0.000, E1   +65.179, E3 +134815.393}
SPL {X   -93.259, Y  +255.690, Z    +0.000, E1   +54.095, E3 +134930.775}
ENDSPLINE

SPLINE
SPL {X  -130.811, Y  +293.568, Z    +0.000, E1   +46.951, E3 +135074.636}
SPL {X  -151.580, Y  +334.479, Z    +0.000, E1   +34.520, E3 +135098.758}
SPL {X  -157.897, Y  +359.846, Z    +0.000, E1   +21.040, E3 +135104.716}
SPL {X  -159.671, Y  +375.443, Z    +0.000, E1   +10.084, E3 +135106.532}
SPL {X  -160.000, Y  +387.403, Z    +0.000, E1    +0.377, E3 +135107.007}
SPL {X  -160.000, Y  +391.807, Z    +0.000, E1    -7.102, E3 +135107.111}
SPL {X  -160.000, Y  +398.244, Z    +0.000, E1   -19.803, E3 +135107.545}
SPL {X  -160.000, Y  +410.795, Z    +0.000, E1   -41.112, E3 +135109.358}
SPL {X  -160.000, Y  +461.796, Z    +0.000, E1   -65.564, E3 +135126.001}
SPL {X  -160.000, Y  +623.854, Z    +0.000, E1   -69.845, E3 +135220.073}
SPL {X  -160.000, Y  +641.581, Z    +0.000, E1   -69.837, E3 +135233.913}
SPL {X  -160.000, Y  +657.932, Z    +0.000, E1   -69.833, E3 +135246.671}
SPL {X  -159.989, Y  +676.310, Z    +0.000, E1   -69.844, E3 +135260.979}
SPL {X  -158.945, Y  +692.747, Z    +0.000, E1   -69.717, E3 +135274.907}
SPL {X  -156.998, Y  +705.248, Z    +0.000, E1   -69.481, E3 +135286.694}
SPL {X  -153.152, Y  +720.707, Z    +0.000, E1   -69.072, E3 +135302.606}
SPL {X  -148.823, Y  +733.152, Z    +0.000, E1   -68.450, E3 +135316.764}
SPL {X  -145.304, Y  +741.384, Z    +0.000, E1   -67.989, E3 +135326.564}
SPL {X  -141.481, Y  +749.119, Z    +0.000, E1   -67.448, E3 +135336.189}
SPL {X  -137.717, Y  +755.849, Z    +0.000, E1   -66.896, E3 +135344.823}
SPL {X  -133.615, Y  +762.417, Z    +0.000, E1   -66.275, E3 +135353.438}
SPL {X  -128.952, Y  +769.117, Z    +0.000, E1   -65.522, E3 +135362.400}
SPL {X  -125.615, Y  +773.501, Z    +0.000, E1   -64.909, E3 +135368.336}
SPL {X   -93.482, Y  +804.250, Z    +0.000, E1   -52.853, E3 +135505.534}
ENDSPLINE

SPLINE
SPL {X  -137.039, Y  +756.986, Z    +0.000, E1   -45.206, E3 +135636.197}
SPL {X  -152.094, Y  +724.074, Z    +0.000, E1   -34.132, E3 +135652.144}
SPL {X  -158.930, Y  +692.872, Z    +0.000, E1   -16.505, E3 +135658.460}
SPL {X  -160.000, Y  +673.072, Z    +0.000, E1    -0.858, E3 +135659.770}
SPL {X  -160.000, Y  +670.505, Z    +0.000, E1    +2.991, E3 +135659.806}
SPL {X  -160.000, Y  +665.157, Z    +0.000, E1   +13.199, E3 +135660.036}
SPL {X  -160.000, Y  +657.552, Z    +0.000, E1   +28.428, E3 +135660.721}
SPL {X  -160.000, Y  +642.088, Z    +0.000, E1   +49.428, E3 +135663.711}
SPL {X  -160.000, Y  +582.331, Z    +0.000, E1   +67.139, E3 +135686.178}
SPL {X  -160.000, Y  +443.344, Z    +0.000, E1   +69.515, E3 +135770.664}
SPL {X  -160.000, Y  +423.295, Z    +0.000, E1   +69.546, E3 +135786.484}
SPL {X  -155.937, Y  +349.874, Z    +0.000, E1   +73.941, E3 +135794.555}
SPL {X  -155.646, Y  +348.628, Z    +0.000, E1   +73.073, E3 +135804.438}
SPL {X  -155.163, Y  +346.655, Z    +0.000, E1   +71.976, E3 +135816.425}
SPL {X  -154.105, Y  +342.669, Z    +0.000, E1   +70.814, E3 +135829.931}
SPL {X  -152.951, Y  +338.733, Z    +0.000, E1   +69.529, E3 +135843.774}
SPL {X  -150.673, Y  +331.871, Z    +0.000, E1   +68.778, E3 +135855.022}
SPL {X  -146.876, Y  +322.238, Z    +0.000, E1   +68.294, E3 +135866.203}
SPL {X  -142.952, Y  +313.834, Z    +0.000, E1   +67.744, E3 +135876.482}
SPL {X  -139.245, Y  +306.891, Z    +0.000, E1   +67.208, E3 +135885.266}
SPL {X  -135.108, Y  +299.992, Z    +0.000, E1   +66.599, E3 +135894.217}
SPL {X  -130.642, Y  +293.328, Z    +0.000, E1   +65.888, E3 +135903.069}
SPL {X  -126.461, Y  +287.682, Z    +0.000, E1   +65.179, E3 +135910.632}
SPL {X   -93.259, Y  +255.690, Z    +0.000, E1   +54.095, E3 +136026.014}
ENDSPLINE

SPLINE
SPL {X  -130.811, Y  +293.568, Z    +0.000, E1   +46.951, E3 +136169.874}
SPL {X  -151.580, Y  +334.479, Z    +0.000, E1   +34.520, E3 +136193.997}
SPL {X  -157.897, Y  +359.846, Z    +0.000, E1   +21.040, E3 +136199.955}
SPL {X  -159.671, Y  +375.443, Z    +0.000, E1   +10.084, E3 +136201.770}
SPL {X  -160.000, Y  +387.403, Z    +0.000, E1    +0.377, E3 +136202.246}
SPL {X  -160.000, Y  +391.807, Z    +0.000, E1    -7.102, E3 +136202.350}
SPL {X  -160.000, Y  +398.244, Z    +0.000, E1   -19.803, E3 +136202.784}
SPL {X  -160.000, Y  +410.795, Z    +0.000, E1   -41.112, E3 +136204.597}
SPL {X  -160.000, Y  +461.796, Z    +0.000, E1   -65.564, E3 +136221.239}
SPL {X  -160.000, Y  +623.854, Z    +0.000, E1   -69.845, E3 +136315.312}
SPL {X  -160.000, Y  +641.581, Z    +0.000, E1   -69.837, E3 +136329.151}
SPL {X  -160.000, Y  +657.932, Z    +0.000, E1   -69.833, E3 +136341.910}
SPL {X  -159.989, Y  +676.310, Z    +0.000, E1   -69.844, E3 +136356.218}
SPL {X  -158.945, Y  +692.747, Z    +0.000, E1   -69.717, E3 +136370.146}
SPL {X  -156.998, Y  +705.248, Z    +0.000, E1   -69.481, E3 +136381.933}
SPL {X  -153.152, Y  +720.707, Z    +0.000, E1   -69.072, E3 +136397.844}
SPL {X  -148.823, Y  +733.152, Z    +0.000, E1   -68.450, E3 +136412.003}
SPL {X  -145.304, Y  +741.384, Z    +0.000, E1   -67.989, E3 +136421.803}
SPL {X  -141.481, Y  +749.119, Z    +0.000, E1   -67.448, E3 +136431.428}
SPL {X  -137.717, Y  +755.849, Z    +0.000, E1   -66.896, E3 +136440.062}
SPL {X  -133.615, Y  +762.417, Z    +0.000, E1   -66.275, E3 +136448.677}
SPL {X  -128.952, Y  +769.117, Z    +0.000, E1   -65.522, E3 +136457.638}
SPL {X  -125.615, Y  +773.501, Z    +0.000, E1   -64.909, E3 +136463.575}
SPL {X   -93.482, Y  +804.250, Z    +0.000, E1   -52.853, E3 +136600.773}
ENDSPLINE

SPLINE
SPL {X  -137.039, Y  +756.986, Z    +0.000, E1   -45.206, E3 +136731.436}
SPL {X  -152.094, Y  +724.074, Z    +0.000, E1   -34.132, E3 +136747.383}
SPL {X  -158.930, Y  +692.872, Z    +0.000, E1   -16.505, E3 +136753.698}
SPL {X  -160.000, Y  +673.072, Z    +0.000, E1    -0.858, E3 +136755.009}
SPL {X  -160.000, Y  +670.505, Z    +0.000, E1    +2.991, E3 +136755.045}
SPL {X  -160.000, Y  +665.157, Z    +0.000, E1   +13.199, E3 +136755.275}
SPL {X  -160.000, Y  +657.552, Z    +0.000, E1   +28.428, E3 +136755.960}
SPL {X  -160.000, Y  +642.088, Z    +0.000, E1   +49.428, E3 +136758.950}
SPL {X  -160.000, Y  +582.331, Z    +0.000, E1   +67.139, E3 +136781.417}
SPL {X  -160.000, Y  +443.344, Z    +0.000, E1   +69.515, E3 +136865.903}
SPL {X  -160.000, Y  +423.295, Z    +0.000, E1   +69.546, E3 +136881.723}
SPL {X  -155.937, Y  +349.874, Z    +0.000, E1   +73.941, E3 +136889.794}
SPL {X  -155.646, Y  +348.628, Z    +0.000, E1   +73.073, E3 +136899.677}
SPL {X  -155.163, Y  +346.655, Z    +0.000, E1   +71.976, E3 +136911.664}
SPL {X  -154.105, Y  +342.669, Z    +0.000, E1   +70.814, E3 +136925.169}
SPL {X  -152.951, Y  +338.733, Z    +0.000, E1   +69.529, E3 +136939.013}
SPL {X  -150.673, Y  +331.871, Z    +0.000, E1   +68.778, E3 +136950.261}
SPL {X  -146.876, Y  +322.238, Z    +0.000, E1   +68.294, E3 +136961.442}
SPL {X  -142.952, Y  +313.834, Z    +0.000, E1   +67.744, E3 +136971.721}
SPL {X  -139.245, Y  +306.891, Z    +0.000, E1   +67.208, E3 +136980.504}
SPL {X  -135.108, Y  +299.992, Z    +0.000, E1   +66.599, E3 +136989.456}
SPL {X  -130.642, Y  +293.328, Z    +0.000, E1   +65.888, E3 +136998.308}
SPL {X  -126.461, Y  +287.682, Z    +0.000, E1   +65.179, E3 +137005.871}
SPL {X   -93.259, Y  +255.690, Z    +0.000, E1   +54.095, E3 +137121.253}
ENDSPLINE

SPLINE
SPL {X  -130.811, Y  +293.568, Z    +0.000, E1   +46.951, E3 +137265.113}
SPL {X  -151.580, Y  +334.479, Z    +0.000, E1   +34.520, E3 +137289.236}
SPL {X  -157.897, Y  +359.846, Z    +0.000, E1   +21.040, E3 +137295.194}
SPL {X  -159.671, Y  +375.443, Z    +0.000, E1   +10.084, E3 +137297.009}
SPL {X  -160.000, Y  +387.403, Z    +0.000, E1    +0.377, E3 +137297.484}
SPL {X  -160.000, Y  +391.807, Z    +0.000, E1    -7.102, E3 +137297.589}
SPL {X  -160.000, Y  +398.244, Z    +0.000, E1   -19.803, E3 +137298.022}
SPL {X  -160.000, Y  +410.795, Z    +0.000, E1   -41.112, E3 +137299.835}
SPL {X  -160.000, Y  +461.796, Z    +0.000, E1   -65.564, E3 +137316.478}
SPL {X  -160.000, Y  +623.854, Z    +0.000, E1   -69.845, E3 +137410.551}
SPL {X  -160.000, Y  +641.581, Z    +0.000, E1   -69.837, E3 +137424.390}
SPL {X  -160.000, Y  +657.932, Z    +0.000, E1   -69.833, E3 +137437.148}
SPL {X  -159.989, Y  +676.310, Z    +0.000, E1   -69.844, E3 +137451.457}
SPL {X  -158.945, Y  +692.747, Z    +0.000, E1   -69.717, E3 +137465.384}
SPL {X  -156.998, Y  +705.248, Z    +0.000, E1   -69.481, E3 +137477.171}
SPL {X  -153.152, Y  +720.707, Z    +0.000, E1   -69.072, E3 +137493.083}
SPL {X  -148.823, Y  +733.152, Z    +0.000, E1   -68.450, E3 +137507.242}
SPL {X  -145.304, Y  +741.384, Z    +0.000, E1   -67.989, E3 +137517.042}
SPL {X  -141.481, Y  +749.119, Z    +0.000, E1   -67.448, E3 +137526.666}
SPL {X  -137.717, Y  +755.849, Z    +0.000, E1   -66.896, E3 +137535.301}
SPL {X  -133.615, Y  +762.417, Z    +0.000, E1   -66.275, E3 +137543.915}
SPL {X  -128.952, Y  +769.117, Z    +0.000, E1   -65.522, E3 +137552.877}
SPL {X  -125.615, Y  +773.501, Z    +0.000, E1   -64.909, E3 +137558.814}
SPL {X   -93.482, Y  +804.250, Z    +0.000, E1   -52.853, E3 +137696.011}
ENDSPLINE

SPLINE
SPL {X  -137.039, Y  +756.986, Z    +0.000, E1   -45.206, E3 +137826.674}
SPL {X  -152.094, Y  +724.074, Z    +0.000, E1   -34.132, E3 +137842.621}
SPL {X  -158.930, Y  +692.872, Z    +0.000, E1   -16.505, E3 +137848.937}
SPL {X  -160.000, Y  +673.072, Z    +0.000, E1    -0.858, E3 +137850.247}
SPL {X  -160.000, Y  +670.505, Z    +0.000, E1    +2.991, E3 +137850.284}
SPL {X  -160.000, Y  +665.157, Z    +0.000, E1   +13.199, E3 +137850.513}
SPL {X  -160.000, Y  +657.552, Z    +0.000, E1   +28.428, E3 +137851.199}
SPL {X  -160.000, Y  +642.088, Z    +0.000, E1   +49.428, E3 +137854.189}
SPL {X  -160.000, Y  +582.331, Z    +0.000, E1   +67.139, E3 +137876.655}
SPL {X  -160.000, Y  +443.344, Z    +0.000, E1   +69.515, E3 +137961.142}
SPL {X  -160.000, Y  +423.295, Z    +0.000, E1   +69.546, E3 +137976.962}
SPL {X  -155.937, Y  +349.874, Z    +0.000, E1   +73.941, E3 +137985.032}
SPL {X  -155.646, Y  +348.628, Z    +0.000, E1   +73.073, E3 +137994.915}
SPL {X  -155.163, Y  +346.655, Z    +0.000, E1   +71.976, E3 +138006.903}
SPL {X  -154.105, Y  +342.669, Z    +0.000, E1   +70.814, E3 +138020.408}
SPL {X  -152.951, Y  +338.733, Z    +0.000, E1   +69.529, E3 +138034.251}
SPL {X  -150.673, Y  +331.871, Z    +0.000, E1   +68.778, E3 +138045.499}
SPL {X  -146.876, Y  +322.238, Z    +0.000, E1   +68.294, E3 +138056.680}
SPL {X  -142.952, Y  +313.834, Z    +0.000, E1   +67.744, E3 +138066.959}
SPL {X  -139.245, Y  +306.891, Z    +0.000, E1   +67.208, E3 +138075.743}
SPL {X  -135.108, Y  +299.992, Z    +0.000, E1   +66.599, E3 +138084.694}
SPL {X  -130.642, Y  +293.328, Z    +0.000, E1   +65.888, E3 +138093.547}
SPL {X  -126.461, Y  +287.682, Z    +0.000, E1   +65.179, E3 +138101.110}
SPL {X   -93.259, Y  +255.690, Z    +0.000, E1   +54.095, E3 +138216.491}
ENDSPLINE

SPLINE
SPL {X  -130.811, Y  +293.568, Z    +0.000, E1   +46.951, E3 +138360.352}
SPL {X  -151.580, Y  +334.479, Z    +0.000, E1   +34.520, E3 +138384.475}
SPL {X  -157.897, Y  +359.846, Z    +0.000, E1   +21.040, E3 +138390.432}
SPL {X  -159.671, Y  +375.443, Z    +0.000, E1   +10.084, E3 +138392.248}
SPL {X  -160.000, Y  +387.403, Z    +0.000, E1    +0.377, E3 +138392.723}
SPL {X  -160.000, Y  +391.807, Z    +0.000, E1    -7.102, E3 +138392.827}
SPL {X  -160.000, Y  +398.244, Z    +0.000, E1   -19.803, E3 +138393.261}
SPL {X  -160.000, Y  +410.795, Z    +0.000, E1   -41.112, E3 +138395.074}
SPL {X  -160.000, Y  +461.796, Z    +0.000, E1   -65.564, E3 +138411.717}
SPL {X  -160.000, Y  +623.854, Z    +0.000, E1   -69.845, E3 +138505.789}
SPL {X  -160.000, Y  +641.581, Z    +0.000, E1   -69.837, E3 +138519.629}
SPL {X  -160.000, Y  +657.932, Z    +0.000, E1   -69.833, E3 +138532.387}
SPL {X  -159.989, Y  +676.310, Z    +0.000, E1   -69.844, E3 +138546.695}
SPL {X  -158.945, Y  +692.747, Z    +0.000, E1   -69.717, E3 +138560.623}
SPL {X  -156.998, Y  +705.248, Z    +0.000, E1   -69.481, E3 +138572.410}
SPL {X  -153.152, Y  +720.707, Z    +0.000, E1   -69.072, E3 +138588.322}
SPL {X  -148.823, Y  +733.152, Z    +0.000, E1   -68.450, E3 +138602.480}
SPL {X  -145.304, Y  +741.384, Z    +0.000, E1   -67.989, E3 +138612.280}
SPL {X  -141.481, Y  +749.119, Z    +0.000, E1   -67.448, E3 +138621.905}
SPL {X  -137.717, Y  +755.849, Z    +0.000, E1   -66.896, E3 +138630.539}
SPL {X  -133.615, Y  +762.417, Z    +0.000, E1   -66.275, E3 +138639.154}
SPL {X  -128.952, Y  +769.117, Z    +0.000, E1   -65.522, E3 +138648.116}
SPL {X  -125.615, Y  +773.501, Z    +0.000, E1   -64.909, E3 +138654.052}
SPL {X   -93.482, Y  +804.250, Z    +0.000, E1   -52.853, E3 +138791.250}
ENDSPLINE

SPLINE
SPL {X  -137.039, Y  +756.986, Z    +0.000, E1   -45.206, E3 +138921.913}
SPL {X  -152.094, Y  +724.074, Z    +0.000, E1   -34.132, E3 +138937.860}
SPL {X  -158.930, Y  +692.872, Z    +0.000, E1   -16.505, E3 +138944.176}
SPL {X  -160.000, Y  +673.072, Z    +0.000, E1    -0.858, E3 +138945.486}
SPL {X  -160.000, Y  +670.505, Z    +0.000, E1    +2.991, E3 +138945.522}
SPL {X  -160.000, Y  +665.157, Z    +0.000, E1   +13.199, E3 +138945.752}
SPL {X  -160.000, Y  +657.552, Z    +0.000, E1   +28.428, E3 +138946.437}
SPL {X  -160.000, Y  +642.088, Z    +0.000, E1   +49.428, E3 +138949.427}
SPL {X  -160.000, Y  +582.331, Z    +0.000, E1   +67.139, E3 +138971.894}
SPL {X  -160.000, Y  +443.344, Z    +0.000, E1   +69.515, E3 +139056.380}
SPL {X  -160.000, Y  +423.295, Z    +0.000, E1   +69.546, E3 +139072.201}
SPL {X  -155.937, Y  +349.874, Z    +0.000, E1   +73.941, E3 +139080.271}
SPL {X  -155.646, Y  +348.628, Z    +0.000, E1   +73.073, E3 +139090.154}
SPL {X  -155.163, Y  +346.655, Z    +0.000, E1   +71.976, E3 +139102.142}
SPL {X  -154.105, Y  +342.669, Z    +0.000, E1   +70.814, E3 +139115.647}
SPL {X  -152.951, Y  +338.733, Z    +0.000, E1   +69.529, E3 +139129.490}
SPL {X  -150.673, Y  +331.871, Z    +0.000, E1   +68.778, E3 +139140.738}
SPL {X  -146.876, Y  +322.238, Z    +0.000, E1   +68.294, E3 +139151.919}
SPL {X  -142.952, Y  +313.834, Z    +0.000, E1   +67.744, E3 +139162.198}
SPL {X  -139.245, Y  +306.891, Z    +0.000, E1   +67.208, E3 +139170.982}
SPL {X  -135.108, Y  +299.992, Z    +0.000, E1   +66.599, E3 +139179.933}
SPL {X  -130.642, Y  +293.328, Z    +0.000, E1   +65.888, E3 +139188.785}
SPL {X  -126.461, Y  +287.682, Z    +0.000, E1   +65.179, E3 +139196.348}
SPL {X   -93.259, Y  +255.690, Z    +0.000, E1   +54.095, E3 +139311.730}
ENDSPLINE

SPLINE
SPL {X  -130.811, Y  +293.568, Z    +0.000, E1   +46.951, E3 +139455.591}
SPL {X  -151.580, Y  +334.479, Z    +0.000, E1   +34.520, E3 +139479.713}
SPL {X  -157.897, Y  +359.846, Z    +0.000, E1   +21.040, E3 +139485.671}
SPL {X  -159.671, Y  +375.443, Z    +0.000, E1   +10.084, E3 +139487.486}
SPL {X  -160.000, Y  +387.403, Z    +0.000, E1    +0.377, E3 +139487.962}
SPL {X  -160.000, Y  +391.807, Z    +0.000, E1    -7.102, E3 +139488.066}
SPL {X  -160.000, Y  +398.244, Z    +0.000, E1   -19.803, E3 +139488.500}
SPL {X  -160.000, Y  +410.795, Z    +0.000, E1   -41.112, E3 +139490.313}
SPL {X  -160.000, Y  +461.796, Z    +0.000, E1   -65.564, E3 +139506.955}
SPL {X  -160.000, Y  +623.854, Z    +0.000, E1   -69.845, E3 +139601.028}
SPL {X  -160.000, Y  +641.581, Z    +0.000, E1   -69.837, E3 +139614.867}
SPL {X  -160.000, Y  +657.932, Z    +0.000, E1   -69.833, E3 +139627.626}
SPL {X  -159.989, Y  +676.310, Z    +0.000, E1   -69.844, E3 +139641.934}
SPL {X  -158.945, Y  +692.747, Z    +0.000, E1   -69.717, E3 +139655.862}
SPL {X  -156.998, Y  +705.248, Z    +0.000, E1   -69.481, E3 +139667.649}
SPL {X  -153.152, Y  +720.707, Z    +0.000, E1   -69.072, E3 +139683.560}
SPL {X  -148.823, Y  +733.152, Z    +0.000, E1   -68.450, E3 +139697.719}
SPL {X  -145.304, Y  +741.384, Z    +0.000, E1   -67.989, E3 +139707.519}
SPL {X  -141.481, Y  +749.119, Z    +0.000, E1   -67.448, E3 +139717.144}
SPL {X  -137.717, Y  +755.849, Z    +0.000, E1   -66.896, E3 +139725.778}
SPL {X  -133.615, Y  +762.417, Z    +0.000, E1   -66.275, E3 +139734.393}
SPL {X  -128.952, Y  +769.117, Z    +0.000, E1   -65.522, E3 +139743.354}
SPL {X  -125.615, Y  +773.501, Z    +0.000, E1   -64.909, E3 +139749.291}
SPL {X   -93.482, Y  +804.250, Z    +0.000, E1   -52.853, E3 +139886.489}
ENDSPLINE

SPLINE
SPL {X  -137.039, Y  +756.986, Z    +0.000, E1   -45.206, E3 +140017.152}
SPL {X  -152.094, Y  +724.074, Z    +0.000, E1   -34.132, E3 +140033.099}
SPL {X  -158.930, Y  +692.872, Z    +0.000, E1   -16.505, E3 +140039.414}
SPL {X  -160.000, Y  +673.072, Z    +0.000, E1    -0.858, E3 +140040.725}
SPL {X  -160.000, Y  +670.505, Z    +0.000, E1    +2.991, E3 +140040.761}
SPL {X  -160.000, Y  +665.157, Z    +0.000, E1   +13.199, E3 +140040.991}
SPL {X  -160.000, Y  +657.552, Z    +0.000, E1   +28.428, E3 +140041.676}
SPL {X  -160.000, Y  +642.088, Z    +0.000, E1   +49.428, E3 +140044.666}
SPL {X  -160.000, Y  +582.331, Z    +0.000, E1   +67.139, E3 +140067.133}
SPL {X  -160.000, Y  +443.344, Z    +0.000, E1   +69.515, E3 +140151.619}
SPL {X  -160.000, Y  +423.295, Z    +0.000, E1   +69.546, E3 +140167.439}
SPL {X  -155.937, Y  +349.874, Z    +0.000, E1   +73.941, E3 +140175.510}
SPL {X  -155.646, Y  +348.628, Z    +0.000, E1   +73.073, E3 +140185.393}
SPL {X  -155.163, Y  +346.655, Z    +0.000, E1   +71.976, E3 +140197.380}
SPL {X  -154.105, Y  +342.669, Z    +0.000, E1   +70.814, E3 +140210.885}
SPL {X  -152.951, Y  +338.733, Z    +0.000, E1   +69.529, E3 +140224.729}
SPL {X  -150.673, Y  +331.871, Z    +0.000, E1   +68.778, E3 +140235.977}
SPL {X  -146.876, Y  +322.238, Z    +0.000, E1   +68.294, E3 +140247.158}
SPL {X  -142.952, Y  +313.834, Z    +0.000, E1   +67.744, E3 +140257.437}
SPL {X  -139.245, Y  +306.891, Z    +0.000, E1   +67.208, E3 +140266.220}
SPL {X  -135.108, Y  +299.992, Z    +0.000, E1   +66.599, E3 +140275.172}
SPL {X  -130.642, Y  +293.328, Z    +0.000, E1   +65.888, E3 +140284.024}
SPL {X  -126.461, Y  +287.682, Z    +0.000, E1   +65.179, E3 +140291.587}
SPL {X   -93.259, Y  +255.690, Z    +0.000, E1   +54.095, E3 +140406.969}
ENDSPLINE

SPLINE
SPL {X  -130.811, Y  +293.568, Z    +0.000, E1   +46.951, E3 +140550.829}
SPL {X  -151.580, Y  +334.479, Z    +0.000, E1   +34.520, E3 +140574.952}
SPL {X  -157.897, Y  +359.846, Z    +0.000, E1   +21.040, E3 +140580.910}
SPL {X  -159.671, Y  +375.443, Z    +0.000, E1   +10.084, E3 +140582.725}
SPL {X  -160.000, Y  +387.403, Z    +0.000, E1    +0.377, E3 +140583.200}
SPL {X  -160.000, Y  +391.807, Z    +0.000, E1    -7.102, E3 +140583.305}
SPL {X  -160.000, Y  +398.244, Z    +0.000, E1   -19.803, E3 +140583.738}
SPL {X  -160.000, Y  +410.795, Z    +0.000, E1   -41.112, E3 +140585.551}
SPL {X  -160.000, Y  +461.796, Z    +0.000, E1   -65.564, E3 +140602.194}
SPL {X  -160.000, Y  +623.854, Z    +0.000, E1   -69.845, E3 +140696.267}
SPL {X  -160.000, Y  +641.581, Z    +0.000, E1   -69.837, E3 +140710.106}
SPL {X  -160.000, Y  +657.932, Z    +0.000, E1   -69.833, E3 +140722.864}
SPL {X  -159.989, Y  +676.310, Z    +0.000, E1   -69.844, E3 +140737.173}
SPL {X  -158.945, Y  +692.747, Z    +0.000, E1   -69.717, E3 +140751.100}
SPL {X  -156.998, Y  +705.248, Z    +0.000, E1   -69.481, E3 +140762.887}
SPL {X  -153.152, Y  +720.707, Z    +0.000, E1   -69.072, E3 +140778.799}
SPL {X  -148.823, Y  +733.152, Z    +0.000, E1   -68.450, E3 +140792.958}
SPL {X  -145.304, Y  +741.384, Z    +0.000, E1   -67.989, E3 +140802.758}
SPL {X  -141.481, Y  +749.119, Z    +0.000, E1   -67.448, E3 +140812.382}
SPL {X  -137.717, Y  +755.849, Z    +0.000, E1   -66.896, E3 +140821.017}
SPL {X  -133.615, Y  +762.417, Z    +0.000, E1   -66.275, E3 +140829.631}
SPL {X  -128.952, Y  +769.117, Z    +0.000, E1   -65.522, E3 +140838.593}
SPL {X  -125.615, Y  +773.501, Z    +0.000, E1   -64.909, E3 +140844.530}
SPL {X   -93.482, Y  +804.250, Z    +0.000, E1   -52.853, E3 +140981.727}
ENDSPLINE

